# B&R Automation Studio project Sorting_Machine_DT
Automation Studio 4.9.2.46; technology packages: Acp10Arnc0 5.12.2, mappView 5.12.1

## Configuration Config1

CPU X20CP1584, AutomationRuntime C4.90, Build 4.1.2, Safety 0.0, Vc V4.72.2

### Task classes (Cpu.sw)
```
Cyclic#1 (cycle 2000 us, tolerance 0 us):
  X_AXIS_M <- XYZ_MANIPULATOR.X_AXIS_M.prg
  Y_AXIS_M <- XYZ_MANIPULATOR.Y_AXIS_M.prg
  Z_AXIS_M <- XYZ_MANIPULATOR.Z_AXIS_M.prg
  X_AXIS_CC <- CAMERA_CONVEYOR.X_AXIS_CC.prg
Cyclic#2 (cycle 10000 us, tolerance 10000 us):
  Main <- Main_Control.Main.prg
DataObjects: Acp10sys
NcDataObjects: acp10etxen <- Motion_Package.acp10etxen.dob, gAxis01_Xa <- Motion_Package.gAxis01_Xobj.gAxis01_Xa.dob, gAxis01_Xi <- Motion_Package.gAxis01_Xobj.gAxis01_Xi.dob, gAxis01_Ya <- Motion_Package.gAxis01_Yobj.gAxis01_Ya.dob, gAxis01_Yi <- Motion_Package.gAxis01_Yobj.gAxis01_Yi.dob, gAxis01_Za <- Motion_Package.gAxis01_Zobj.gAxis01_Za.dob, gAxis01_Zi <- Motion_Package.gAxis01_Zobj.gAxis01_Zi.dob, gAxis01_Ca <- Motion_Package.gAxis01_Cobj.gAxis01_Ca.dob, gAxis01_Ci <- Motion_Package.gAxis01_Cobj.gAxis01_Ci.dob
Binaries: udbdef, arsvcreg, FWRules, mvLoader, TCData, acp10cfg, Acp10map, iomap, asfw, Role, Config, sysconf, arconfig, ashwd, User, ashwac
Libraries: Acp10man, Acp10par, NcGlobal, Acp10_MC, sys_lib, brsystem, runtime, MpAxis, MpBase, MpCom, rp_funcx, standard, Acp10sim, astime, arssl, asbrstr, fileio, powerlnk, dataobj
```

### Hardware
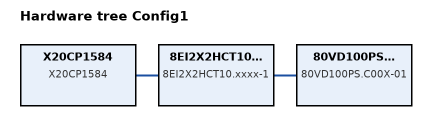
```
80VD100PS.C00X-01 : 80VD100PS.C00X-01 v2.5.0.0  [PLK1 -> 8EI2X2HCT10.xxxx-1.PLK2 (NodeNumber=2) [Cable Type=PowerlinkCable, Length=10, Version=1.0.0.3]]
  MotionTP = Acp10Arnc0
  Simulate = complete
  BothEndSwitchesAreNormallyOpen_r1 = on
  QuickStopIsNormallyOpen_r1 = on
8EI2X2HCT10.xxxx-1 : 8EI2X2HCT10.xxxx-1 v2.3.0.3  [PLK1 -> X20CP1584.IF3 (NodeNumber=1) [Cable Type=PowerlinkCable, Length=10, Version=1.0.0.3]; PLK2 -> 80VD100PS.C00X-01.PLK1 (NodeNumber=1) [Cable Type=PowerlinkCable, Length=10, Version=1.0.0.3]]
  MotionTP = Acp10Arnc0
  Simulate = complete
  BothEndSwitchesAreNormallyOpen_r1 = on
  QuickStopIsNormallyOpen_r1 = on
X20CP1584 : X20CP1584 v1.9.0.0
  Connector IF2:
    ActivateDevice = 1
  ConfigurationID = Sorting_Machine_DT_Config1
  Simulation = 1
  TimerDeviceType = EPLX2X
  TimerDevice = X20CP1584.IF3
  TaskClassIdleTime = 2000
  Cyclic1Duration = 2000
  Cyclic1Tolerance = 0
  Cyclic2Duration = 10000
  Cyclic2Tolerance = 10000
  ActivateOpcUa = 1
  OpcUaInformationModels_PV_Version = 1
```

### OpcUa.uanodeset - X20CP1584/Connectivity/OpcUA/OpcUa.uanodeset
```
UANodeSet:
  NamespaceUris:
    Uri = http://customer.com/mynamespace/
  Aliases:
    Alias = i=1 (Alias=Boolean)
    Alias = i=2 (Alias=SByte)
    Alias = i=3 (Alias=Byte)
    Alias = i=4 (Alias=Int16)
    Alias = i=5 (Alias=UInt16)
    Alias = i=6 (Alias=Int32)
    Alias = i=7 (Alias=UInt32)
    Alias = i=12 (Alias=String)
```

### Acp10cfg.ncc - X20CP1584/Motion/Acp10cfg.ncc
```
NcConfiguration (Version=5.12.2, NcSwId=Acp10)
  ACP10CF1_typ:
    cnt_nettrc_rec_drive = 1500
    bufsize_trace_upload = 1200
    tc_nc_man_task = Cyclic #1
    glob_pv_as_ncobject = Yes
    ncsys_dl_broadcast = Yes
    ncsys_dl_acp_reset = Yes
    safemc_log_err_to_ax = Yes
    network_init:
      ncsw_init_execute = Yes
      automatic_execute = No
      node_nr_warning = Yes
      net_err_before_ncact = Yes
    nettrc:
      enter_parsecrec = Yes
      enter_ncaction = Yes
      save_ring_startidx = Yes
    cam_prof_download:
      cam_dat_dl_parallel = No
      tc_cam_dl_parallel = Task class for NC Manager task
    plk_if[0]:
      if_name = IF3
      tc_CycDat_PLCopen = Task class for NC Manager task
      mc_broadcast_extdat = No
```

### Acp10map.ncm - X20CP1584/Motion/Acp10map.ncm
```
NcMapping (NcSwId=Acp10)
  NcObject gAxis01_X (ModuleId=8EI2X2HCT10.xxxx-1, Type=ncAXIS, Channel=1, AcoposSimulation=Off, InitParameter=gAxis01_Xi, AcoposParameter=gAxis01_Xa, Disabled=FALSE, ModuleDisabled=FALSE)
  NcObject gAxis01_Y (ModuleId=8EI2X2HCT10.xxxx-1, Type=ncAXIS, Channel=2, AcoposSimulation=Off, InitParameter=gAxis01_Yi, AcoposParameter=gAxis01_Ya, Disabled=FALSE, ModuleDisabled=FALSE)
  NcObject gAxis01_Z (ModuleId=8EI2X2HCT10.xxxx-1, Type=ncAXIS, Channel=3, AcoposSimulation=Off, InitParameter=gAxis01_Zi, AcoposParameter=gAxis01_Za, Disabled=FALSE, ModuleDisabled=FALSE)
  NcObject 8EI2X2HCT10.xxxx-1_ncV_AXIS1 (ModuleId=8EI2X2HCT10.xxxx-1, Type=ncV_AXIS, Channel=1, Disabled=TRUE, ModuleDisabled=FALSE)
  NcObject 8EI2X2HCT10.xxxx-1_ncV_AXIS2 (ModuleId=8EI2X2HCT10.xxxx-1, Type=ncV_AXIS, Channel=2, Disabled=TRUE, ModuleDisabled=FALSE)
  NcObject 8EI2X2HCT10.xxxx-1_ncV_AXIS3 (ModuleId=8EI2X2HCT10.xxxx-1, Type=ncV_AXIS, Channel=3, Disabled=TRUE, ModuleDisabled=FALSE)
  NcObject gAxis01_C (ModuleId=80VD100PS.C00X-01, Type=ncAXIS, Channel=1, AcoposSimulation=Off, InitParameter=gAxis01_Ci, AcoposParameter=gAxis01_Ca, Disabled=FALSE, ModuleDisabled=FALSE)
  NcObject 80VD100PS.C00X-01_ncV_AXIS1 (ModuleId=80VD100PS.C00X-01, Type=ncV_AXIS, Channel=1, Disabled=TRUE, ModuleDisabled=FALSE)
```

### Config.mpaxisbasic - X20CP1584/Motion/Config.mpaxisbasic
```
Element gAxisBasic_Axis_M_X (Type=mpaxisbasic)
Element gAxisBasic_Axis_M_Z (Type=mpaxisbasic)
Element gAxisBasic_Axis_M_Y (Type=mpaxisbasic)
Element gAxisBasic_Axis_CC_X (Type=mpaxisbasic)
```

- Safety project (password-protected, skipped)

## Logical view

Binary libraries used (declarations not repeated): operator, runtime, astime, AsIecCon, Acp10man 5.12.2, Acp10par 5.12.2, NcGlobal 5.12.2, Acp10_MC 5.12.2, sys_lib, brsystem, MpAxis 1.75.0, MpBase 5.12.0, MpCom 5.12.0, standard, Acp10sim 5.12.2

### Global.typ - Global data types
```iecst
TYPE
	mapp_view_str : 	STRUCT
		active : BOOL;
		is_homed : BOOL;
		power_on : BOOL;
		cam_obj_id : USINT;
		br_pad_obj_id : ARRAY[0..3]OF USINT;
		smc_pad_obj_id : ARRAY[0..3]OF USINT;
	END_STRUCT;
	object_str : 	STRUCT
		write : object_w_str;
		read : object_r_str;
	END_STRUCT;
	object_w_str : 	STRUCT
		set_object_id : USINT;
		reset : BOOL;
		detach : BOOL;
		attach : BOOL;
	END_STRUCT;
	object_r_str : 	STRUCT
		object_id : USINT;
		object_type : USINT;
	END_STRUCT;
	digT_service_control_str : 	STRUCT
		power : BOOL;
		home : BOOL;
		start : BOOL;
		actual_state : USINT;
		object : object_str;
		mapp_view : mapp_view_str;
	END_STRUCT;
	digT_control_llinp_str : 	STRUCT
		pos : LREAL;
		vel : LREAL;
	END_STRUCT;
	digT_control_linp_enum :
		(
		LINP_CTRL_WAIT_STATE := 0,
		LINP_CTRL_LOAD_PARAM_STATE := 10,
		LINP_CTRL_SET_POSITION_STATE := 11,
		LINP_CTRL_STOP_STATE := 12
		);
	axis_str : 	STRUCT
		actual_velocity : LREAL;
		actual_position : LREAL;
		actual_state : digT_control_linp_enum;
		parameter : digT_control_llinp_str;
		start : BOOL;
		stop : BOOL;
		active : BOOL;
		power_on : BOOL;
		is_homed : BOOL;
	END_STRUCT;
	camera_conv_str : 	STRUCT
		X : axis_str;
	END_STRUCT;
	xyz_manip_str : 	STRUCT
		X : axis_str;
		Y : axis_str;
		Z : axis_str;
	END_STRUCT;
	dt_main_str : 	STRUCT
		camera : camera_str;
		xyz_manipulator : xyz_manip_str;
		camera_conveyor : camera_conv_str;
		service : digT_service_control_str;
	END_STRUCT;
	camera_str : 	STRUCT
		scan : BOOL;
	END_STRUCT;
END_TYPE
```

### Global.var - Global variables
```iecst
VAR
	gAxis01_X : ACP10AXIS_typ;
	gAxis01_Y : ACP10AXIS_typ;
	gAxis01_Z : ACP10AXIS_typ;
	gAxis01_C : ACP10AXIS_typ;
	dT_Main : dt_main_str;
END_VAR
```

### Package Logical/Libraries - Global libraries

### Library Logical/Libraries/rp_funcx (ANSIC)

#### Types.typ - Exported data types
```iecst
TYPE
	default_param_smcT_str : 	STRUCT
		MAX_POSITION : LREAL;
		MIN_POSITION : LREAL;
		MAX_VELOCITY : LREAL;
		MIN_VELOCITY : LREAL;
	END_STRUCT;
	param_lim_struct : 	STRUCT
		velocity : LREAL;
		position_end : LREAL;
		position_start : LREAL;
		mode : limit_sequence_enum;
		time : ARRAY[0..1]OF TIME;
		signal : BOOL;
		signal_inPos : ARRAY[0..1]OF BOOL;
		elapsed_time : ARRAY[0..1]OF TIME;
		time_signal : ARRAY[0..1]OF USINT;
	END_STRUCT;
	parameters_structure_set : 	STRUCT
		position : LREAL;
		velocity : LREAL;
		limit : param_lim_struct;
		sequence : param_sv_struct;
		MAX_VELOCITY : LREAL := 0;
		MIN_VELOCITY : LREAL := 0;
		MAX_POSITION : LREAL := 0;
		MIN_POSITION : LREAL := 0;
		default_parameters : BOOL;
		set_velocity : LREAL;
		set_position : LREAL;
	END_STRUCT;
	parameters_structure_actual : 	STRUCT
		position : LREAL;
		velocity : REAL;
		torque : LREAL;
		motorTemperature : LREAL;
		lagError : LREAL;
		profinet_pos : ARRAY[0..5]OF USINT;
		profinet_vel : ARRAY[0..5]OF USINT;
	END_STRUCT;
	param_sv_struct : 	STRUCT
		position : ARRAY[0..4]OF LREAL;
		velocity : ARRAY[0..4]OF LREAL;
		mode : limit_sequence_enum;
		signal : BOOL;
		time : ARRAY[0..4]OF TIME;
		signal_inPos : ARRAY[0..4]OF BOOL;
		elapsed_time : ARRAY[0..4]OF TIME;
		time_signal : ARRAY[0..4]OF USINT;
	END_STRUCT;
	mode_structure : 	STRUCT
		manual : instruction_structure_manual;
		automatic : instruction_structure_auto;
		stop : BOOL;
		home : BOOL;
		mode : USINT;
	END_STRUCT;
	SMCTrak_enum :
		(
		INITIALIZATION_STATE := 0,
		POWER_STATE := 10,
		HOME_STATE_1 := 20,
		HOME_STATE_2 := 21,
		HOME_STATE_3 := 22,
		WAIT_STATE := 30,
		MOVE_HOME_1 := 35,
		MOVE_HOME_2 := 36,
		AUTO_MODE_STATE_RT_1 := 40,
		AUTO_MODE_STATE_RT_2 := 41,
		AUTO_MODE_STATE_RT_3 := 42,
		AUTO_MODE_STATE_UL_1 := 50,
		AUTO_MODE_STATE_UL_2 := 51,
		AUTO_MODE_STATE_UL_3 := 52,
		AUTO_MODE_STATE_SS_1 := 60,
		AUTO_MODE_STATE_SS_2 := 62,
		MANUAL_MODE_STATE_1 := 70,
		MANUAL_MODE_STATE_2 := 71,
		ERROR_STATE_1 := 100,
		ERROR_STATE_2 := 101,
		ERROR_STATE_3 := 102,
		ERROR_STATE_4 := 103,
		ERROR_STATE_5 := 104
		);
	limit_sequence_enum :
		(
		INSTR_SIGNAL := 0,
		INSTR_TIME := 1
		);
	Internal_structure_SMCtrak : 	STRUCT
		Before_state : SMCTrak_enum;
		State : SMCTrak_enum;
		Local : internal_local_smctrak;
		Timer : internal_smctrak_timer;
	END_STRUCT;
	internal_smctrak_timer : 	STRUCT
		enable_time : BOOL;
		output_time : BOOL;
		wait_time : TIME;
		elapsed_time : {REDUND_UNREPLICABLE} TIME;
	END_STRUCT;
	internal_local_smctrak : 	STRUCT
		set_position : LREAL;
		set_velocity : LREAL;
		before_position : LREAL;
		before_velocity : LREAL;
		sum_position : LREAL;
		sum_velocity : LREAL;
		count_sequence : USINT;
		pos_sequence : LREAL;
	END_STRUCT;
	instruction_structure_manual : 	STRUCT
		start : BOOL;
	END_STRUCT;
	instruction_structure_auto : 	STRUCT
		start : BOOL;
		instruction : automatic_instruction_enum;
	END_STRUCT;
	automatic_instruction_enum :
		(
		INSTR_REAL_TIME := 0,
		INSTR_LOWER_UPPER_LIMIT := 1,
		INSTR_SEQUENCE := 2
		);
END_TYPE
```

#### rp_funcx.fun - Exported functions and function blocks
```iecst
FUNCTION_BLOCK SMC_PAD (*TODO: Add your comment here*) (*$GROUP=User,$CAT=User,$GROUPICON=User.png,$CATICON=User.png*)
	VAR_INPUT
		Enable : {REDUND_UNREPLICABLE} BOOL;
		Power : BOOL;
		Home : BOOL;
		Absolute_Position : LREAL;
		MpAxis : REFERENCE TO MpAxisBasic;
		MpAxisParType : REFERENCE TO MpAxisBasicParType;
		MpAxisCyclic : REFERENCE TO MpAxisCyclicSet;
		MpAxisCyclicParType : REFERENCE TO MpAxisCyclicSetParType;
		Mode : mode_structure;
		Default_parameters : default_param_smcT_str;
		Set_Parameters : parameters_structure_set;
	END_VAR
	VAR_OUTPUT
		Actual_State : SMCTrak_enum;
		PowerOn : BOOL;
		IsHomed : BOOL;
		Actual_Parameters : parameters_structure_actual;
		InPosition : BOOL;
		Active : BOOL;
		Status : DINT;
	END_VAR
	VAR
		Internal : Internal_structure_SMCtrak;
	END_VAR
END_FUNCTION_BLOCK
```

#### SMC_PAD.c
```c
/**
 * MIT License
 * Copyright(c) 2020 Roman Parak
 * Permission is hereby granted, free of charge, to any person obtaining a copy
 * of this software and associated documentation files (the "Software"), to deal
 * in the Software without restriction, including without limitation the rights
 * to use, copy, modify, merge, publish, distribute, sublicense, and/or sell
 * copies of the Software, and to permit persons to whom the Software is
 * furnished to do so, subject to the following conditions:
 * The above copyright notice and this permission notice shall be included in all
 * copies or substantial portions of the Software.
 * THE SOFTWARE IS PROVIDED "AS IS", WITHOUT WARRANTY OF ANY KIND, EXPRESS OR
 * IMPLIED, INCLUDING BUT NOT LIMITED TO THE WARRANTIES OF MERCHANTABILITY,
 * FITNESS FOR A PARTICULAR PURPOSE AND NONINFRINGEMENT. IN NO EVENT SHALL THE
 * AUTHORS OR COPYRIGHT HOLDERS BE LIABLE FOR ANY CLAIM, DAMAGES OR OTHER
 * LIABILITY, WHETHER IN AN ACTION OF CONTRACT, TORT OR OTHERWISE, ARISING FROM,
 * OUT OF OR IN CONNECTION WITH THE SOFTWARE OR THE USE OR OTHER DEALINGS IN THE
 * SOFTWARE.
 */
/**
 * Author   : Roman Parak
 * Email    : Roman.Parak@outlook.com
 * File Name: SMC_PAD.c
 */

#include <bur/plctypes.h>
#include <stdio.h>
#include <stdlib.h>
#include <MpAxis.h>
#include <math.h>
#include <standard.h>

#ifdef __cplusplus
	extern "C"
	{
#endif
#include "rp_funcx.h"
#ifdef __cplusplus
	};
#endif

// ************************************************************************************************************************************ //
// -------------------------------------------------------------  DECLARATIONS -------------------------------------------------------- //
// ************************************************************************************************************************************ //
// Timer
_LOCAL TON_typ ton_1;
// FUNCTION // DECLARATION //
void update_cyclicParameters(struct SMC_PAD* smc_pad, LREAL position, LREAL velocity);
BOOL set_time(BOOL enable, TIME t);
// INITIALIZATION // RESET //
void initialization_smc_pad(struct SMC_PAD* smc_pad);
void reset_parameters(struct SMC_PAD* smc_pad);
void parameters_null(struct SMC_PAD* smc_pad);

// ************************************************************************************************************************************ //
// --------------------------------------------------------------  MAIN --------------------------------------------------------------- //
// ************************************************************************************************************************************ //
void SMC_PAD(struct SMC_PAD* smc_pad)
{
	// *********************************************************//
	// ---------------- INITIALIZATION  ----------------------- //
	// *********************************************************//
	if(smc_pad->Enable != 1){
		initialization_smc_pad(smc_pad);
	}

	// *********************************************************//
	// ---------------- PAD MAIN STATE  ----------------------- //
	// *********************************************************//
	switch(smc_pad->Internal.State){
		case INITIALIZATION_STATE:
			{
				/*************************************** INITIALIZATION STATE ******************************************/
				if((smc_pad->MpAxis->Error != 0 || smc_pad->MpAxisCyclic->Error != 0) || (smc_pad->MpAxis->StatusID != 0 || smc_pad->MpAxisCyclic->StatusID != 0)){
					smc_pad->Internal.Before_state = smc_pad->Internal.State;
					smc_pad->Internal.State 	   = ERROR_STATE_1;
				}

				if(smc_pad->MpAxis->Active == 1 && smc_pad->MpAxisCyclic->Active == 1){
					smc_pad->Active 	    = 1;
					smc_pad->Internal.State = POWER_STATE;
				}else{
					smc_pad->Active = 0;
				}
			}
			break;
		case POWER_STATE:
			{
				/*************************************** POWER STATE ******************************************/
				if((smc_pad->MpAxis->Error != 0 || smc_pad->MpAxisCyclic->Error != 0) || (smc_pad->MpAxis->StatusID != 0 || smc_pad->MpAxisCyclic->StatusID != 0)){
					smc_pad->Internal.Before_state = smc_pad->Internal.State;
					smc_pad->Internal.State 	   = ERROR_STATE_1;
				}

				if(smc_pad->Power == 1){
					// power state
					smc_pad->MpAxis->Power = 1;

					if(smc_pad->MpAxis->PowerOn == 1){
						smc_pad->Internal.State = HOME_STATE_1;
					}
				}
			}
			break;
		case HOME_STATE_1:
			{
				/*************************************** HOME (1) STATE ******************************************/
				if((smc_pad->MpAxis->Error != 0 || smc_pad->MpAxisCyclic->Error != 0) || (smc_pad->MpAxis->StatusID != 0 || smc_pad->MpAxisCyclic->StatusID != 0)){
					smc_pad->Internal.Before_state = smc_pad->Internal.State;
					smc_pad->Internal.State 	   = ERROR_STATE_1;
				}

				if(smc_pad->Home == 1){
					if(smc_pad->MpAxis->Position == 0 || (fabs(smc_pad->MpAxis->Position) == smc_pad->Absolute_Position)){
						// home state
						smc_pad->MpAxis->Home = 1;

						if(smc_pad->MpAxis->IsHomed == 1){
							smc_pad->MpAxis->Home   = 0;
							smc_pad->Internal.State = WAIT_STATE;
						}
					}else{
						smc_pad->Internal.State = HOME_STATE_2;
					}
				}

			}
			break;
		case HOME_STATE_2:
			{
				/*************************************** HOME (2) STATE ******************************************/
				if((smc_pad->MpAxis->Error != 0 || smc_pad->MpAxisCyclic->Error != 0) || (smc_pad->MpAxis->StatusID != 0 || smc_pad->MpAxisCyclic->StatusID != 0)){
					smc_pad->Internal.Before_state = smc_pad->Internal.State;
					smc_pad->Internal.State 	   = ERROR_STATE_1;
				}

				smc_pad->MpAxisParType->Home.Position = fabs(fabs(smc_pad->MpAxis->Position) - smc_pad->Absolute_Position);
				smc_pad->MpAxis->Update = 1;

				if(smc_pad->MpAxis->UpdateDone == 1){
					smc_pad->MpAxis->Update = 0;
					smc_pad->Internal.State = HOME_STATE_3;
				}

			}
			break;
		case HOME_STATE_3:
			{
				/*************************************** HOME (3) STATE ******************************************/
				if((smc_pad->MpAxis->Error != 0 || smc_pad->MpAxisCyclic->Error != 0) || (smc_pad->MpAxis->StatusID != 0 || smc_pad->MpAxisCyclic->StatusID != 0)){
					smc_pad->Internal.Before_state = smc_pad->Internal.State;
					smc_pad->Internal.State 	   = ERROR_STATE_1;
				}

				smc_pad->MpAxis->Home = 1;

				if(smc_pad->MpAxis->IsHomed == 1){
					smc_pad->MpAxis->Home   = 0;
					smc_pad->Internal.State = MOVE_HOME_1;
				}
			}
			break;
		case WAIT_STATE:
			{
				/*************************************** WAIT STATE ******************************************/
				if((smc_pad->MpAxis->Error != 0 || smc_pad->MpAxisCyclic->Error != 0) || (smc_pad->MpAxis->StatusID != 0 || smc_pad->MpAxisCyclic->StatusID != 0)){
					smc_pad->Internal.Before_state = smc_pad->Internal.State;
					smc_pad->Internal.State 	   = ERROR_STATE_1;
				}

				if(smc_pad->Mode.automatic.start == 1){
					smc_pad->MpAxis->Stop = 0;
					smc_pad->Mode.stop    = 0;
					if(smc_pad->Mode.automatic.instruction == INSTR_REAL_TIME){
						// real time {0}
						smc_pad->Internal.State  = AUTO_MODE_STATE_RT_1;
					}else if(smc_pad->Mode.automatic.instruction == INSTR_LOWER_UPPER_LIMIT){
						// upper / lower limit {1}
						// Set time parameters
						int i;
						for(i = 0; i < (int)(sizeof(smc_pad->Set_Parameters.limit.time)/sizeof(smc_pad->Set_Parameters.limit.time[0])); i++){
							if(smc_pad->Set_Parameters.limit.time_signal[i] == 0){
								smc_pad->Set_Parameters.limit.time[i] = 500;
							}else{
								smc_pad->Set_Parameters.limit.time[i] = smc_pad->Set_Parameters.limit.time_signal[0]*500;
							}
						}
						smc_pad->Internal.State  = AUTO_MODE_STATE_UL_1;
					}else if(smc_pad->Mode.automatic.instruction == INSTR_SEQUENCE){
						// sequence of steps {2}
						// Set time parameters
						int i;
						for(i = 0; i < (int)(sizeof(smc_pad->Set_Parameters.sequence.time)/sizeof(smc_pad->Set_Parameters.sequence.time[0])); i++){
							if(smc_pad->Set_Parameters.sequence.time_signal[i] == 0){
								smc_pad->Set_Parameters.sequence.time[i] = 500;
							}else{
								smc_pad->Set_Parameters.sequence.time[i] = smc_pad->Set_Parameters.sequence.time_signal[0]*500;
							}
						}
						smc_pad->Internal.State  = AUTO_MODE_STATE_SS_1;
					}
				}else if(smc_pad->Mode.manual.start == 1){
					smc_pad->Mode.stop      = 0;
					smc_pad->Internal.State = MANUAL_MODE_STATE_1;
				}else if(smc_pad->Mode.home == 1){
					if(smc_pad->MpAxisCyclic->Info.SlavePosition != 0){
						smc_pad->Internal.State = MOVE_HOME_1;
					}
				}else{
					smc_pad->Mode.stop = 0;
				}
			}
			break;
		case MOVE_HOME_1:
			{
				/*************************************** MOVE HOME (1) STATE ******************************************/
				if((smc_pad->MpAxis->Error != 0 || smc_pad->MpAxisCyclic->Error != 0) || (smc_pad->MpAxis->StatusID != 0 || smc_pad->MpAxisCyclic->StatusID != 0)){
					smc_pad->Internal.Before_state = smc_pad->Internal.State;
					smc_pad->Internal.State 	   = ERROR_STATE_1;
				}

				update_cyclicParameters(smc_pad, smc_pad->MpAxisCyclic->Info.SlavePosition, (smc_pad->Set_Parameters.MIN_VELOCITY*30));

				smc_pad->MpAxisCyclic->Update = 1;

				if(smc_pad->MpAxisCyclic->UpdateDone == 1){
					smc_pad->MpAxisCyclic->Update = 0;
					smc_pad->Internal.State       = MOVE_HOME_2;
				}
			}
			break;
		case MOVE_HOME_2:
			{
				/*************************************** MOVE HOME (2) STATE ******************************************/
				if((smc_pad->MpAxis->Error != 0 || smc_pad->MpAxisCyclic->Error != 0) || (smc_pad->MpAxis->StatusID != 0 || smc_pad->MpAxisCyclic->StatusID != 0)){
					smc_pad->Internal.Before_state = smc_pad->Internal.State;
					smc_pad->Internal.State 	   = ERROR_STATE_1;
				}

				if(smc_pad->MpAxisCyclic->CyclicPosition == 0){
					smc_pad->MpAxisCyclic->CyclicPosition = 1;
				}

				smc_pad->MpAxisCyclic->Position = smc_pad->Set_Parameters.MIN_POSITION;

				if(smc_pad->MpAxisCyclic->Info.SlavePosition == 0){
					smc_pad->Mode.home      = 0;
					smc_pad->Internal.State = WAIT_STATE;
				}
			}
			break;
		case AUTO_MODE_STATE_RT_1:
			{
				/*************************************** AUTO MODE Real-Time (1) STATE ******************************************/
				if((smc_pad->MpAxis->Error != 0 || smc_pad->MpAxisCyclic->Error != 0) || (smc_pad->MpAxis->StatusID != 0 || smc_pad->MpAxisCyclic->StatusID != 0)){
					smc_pad->Internal.Before_state = smc_pad->Internal.State;
					smc_pad->Internal.State 	   = ERROR_STATE_1;
				}

				if(smc_pad->Set_Parameters.position != smc_pad->Internal.Local.before_position){
					smc_pad->MpAxisCyclic->Position 	 = smc_pad->Set_Parameters.position;
					smc_pad->Internal.Local.set_position = smc_pad->Set_Parameters.position;
					smc_pad->Internal.Local.set_velocity = smc_pad->Set_Parameters.velocity;

					if((fabs(smc_pad->Set_Parameters.position - smc_pad->Internal.Local.before_position) == smc_pad->Internal.Local.sum_position) && (fabs(smc_pad->Set_Parameters.velocity - smc_pad->Internal.Local.before_velocity) == smc_pad->Internal.Local.sum_velocity)){
						smc_pad->Internal.State = AUTO_MODE_STATE_RT_2;
					}else{
						smc_pad->Internal.Local.sum_position  = fabs(smc_pad->Set_Parameters.position - smc_pad->Internal.Local.before_position);
						smc_pad->Internal.Local.sum_velocity  = fabs(smc_pad->Set_Parameters.velocity - smc_pad->Internal.Local.before_velocity);
						smc_pad->Internal.State         	  = AUTO_MODE_STATE_RT_3;
					}
				}
			}
			break;
		case AUTO_MODE_STATE_RT_2:
			{
				/*************************************** AUTO MODE Real-Time (2) STATE ******************************************/
				if((smc_pad->MpAxis->Error != 0 || smc_pad->MpAxisCyclic->Error != 0) || (smc_pad->MpAxis->StatusID != 0 || smc_pad->MpAxisCyclic->StatusID != 0)){
					smc_pad->Internal.Before_state = smc_pad->Internal.State;
					smc_pad->Internal.State 	   = ERROR_STATE_1;
				}

				if(smc_pad->MpAxisCyclic->CyclicPosition == 0){
					smc_pad->MpAxisCyclic->CyclicPosition = 1;
				}

				if(smc_pad->MpAxisCyclic->Info.SlavePosition == smc_pad->Internal.Local.set_position){
					smc_pad->Internal.Local.before_position = smc_pad->Internal.Local.set_position;
					smc_pad->Internal.Local.before_velocity = smc_pad->Internal.Local.set_velocity;
					smc_pad->Internal.State           	    = AUTO_MODE_STATE_RT_1;
				}
			}
			break;
		case AUTO_MODE_STATE_RT_3:
			{
				/*************************************** AUTO MODE Real-Time (3) STATE ******************************************/
				if((smc_pad->MpAxis->Error != 0 || smc_pad->MpAxisCyclic->Error != 0) || (smc_pad->MpAxis->StatusID != 0 || smc_pad->MpAxisCyclic->StatusID != 0)){
					smc_pad->Internal.Before_state = smc_pad->Internal.State;
					smc_pad->Internal.State 	   = ERROR_STATE_1;
				}

				update_cyclicParameters(smc_pad, fabs(smc_pad->Set_Parameters.position - smc_pad->MpAxisCyclic->Info.SlavePosition), smc_pad->Set_Parameters.velocity);

				smc_pad->MpAxisCyclic->Update = 1;

				if(smc_pad->MpAxisCyclic->UpdateDone == 1){
					smc_pad->MpAxisCyclic->Update = 0;
					smc_pad->Internal.State       = AUTO_MODE_STATE_RT_2;
				}
			}
			break;
		case MANUAL_MODE_STATE_1:
			{
				/*************************************** MANUAL MODE (1) STATE ******************************************/
				if((smc_pad->MpAxis->Error != 0 || smc_pad->MpAxisCyclic->Error != 0) || (smc_pad->MpAxis->StatusID != 0 || smc_pad->MpAxisCyclic->StatusID != 0)){
					smc_pad->Internal.Before_state = smc_pad->Internal.State;
					smc_pad->Internal.State 	   = ERROR_STATE_1;
				}

				update_cyclicParameters(smc_pad, smc_pad->Set_Parameters.MAX_POSITION, smc_pad->Set_Parameters.MAX_VELOCITY);

				smc_pad->MpAxisCyclic->Update = 1;

				if(smc_pad->MpAxisCyclic->UpdateDone == 1){
					smc_pad->MpAxisCyclic->Update = 0;
					smc_pad->Internal.State       = MANUAL_MODE_STATE_2;
				}
			}
			break;
		case MANUAL_MODE_STATE_2:
			{
				/*************************************** MANUAL MODE (2) STATE ******************************************/
				if((smc_pad->MpAxis->Error != 0 || smc_pad->MpAxisCyclic->Error != 0) || (smc_pad->MpAxis->StatusID != 0 || smc_pad->MpAxisCyclic->StatusID != 0)){
					smc_pad->Internal.Before_state = smc_pad->Internal.State;
					smc_pad->Internal.State 	   = ERROR_STATE_1;
				}

				if(smc_pad->MpAxisCyclic->CyclicPosition == 0){
					smc_pad->MpAxisCyclic->CyclicPosition = 1;
				}

				smc_pad->MpAxisCyclic->Position = smc_pad->Set_Parameters.position;
			}
			break;
		case AUTO_MODE_STATE_UL_1:
			{
				/*************************************** AUTO MODE Upper/Lower (1) STATE ******************************************/
				if((smc_pad->MpAxis->Error != 0 || smc_pad->MpAxisCyclic->Error != 0) || (smc_pad->MpAxis->StatusID != 0 || smc_pad->MpAxisCyclic->StatusID != 0)){
					smc_pad->Internal.Before_state = smc_pad->Internal.State;
					smc_pad->Internal.State 	   = ERROR_STATE_1;
				}

				update_cyclicParameters(smc_pad, (smc_pad->Set_Parameters.limit.position_start - smc_pad->Set_Parameters.limit.position_end), smc_pad->Set_Parameters.limit.velocity);

				smc_pad->MpAxisCyclic->Update = 1;

				if(smc_pad->MpAxisCyclic->UpdateDone == 1){
					smc_pad->MpAxisCyclic->Update = 0;
					smc_pad->Internal.State       = AUTO_MODE_STATE_UL_2;
				}
			}
			break;
		case AUTO_MODE_STATE_UL_2:
			{
				/*************************************** AUTO MODE Upper/Lower (2) STATE ******************************************/
				if((smc_pad->MpAxis->Error != 0 || smc_pad->MpAxisCyclic->Error != 0) || (smc_pad->MpAxis->StatusID != 0 || smc_pad->MpAxisCyclic->StatusID != 0)){
					smc_pad->Internal.Before_state = smc_pad->Internal.State;
					smc_pad->Internal.State 	   = ERROR_STATE_1;
				}

				if(smc_pad->MpAxisCyclic->CyclicPosition == 0){
					smc_pad->MpAxisCyclic->CyclicPosition = 1;
				}

				if(smc_pad->MpAxisCyclic->Info.SlavePosition != smc_pad->Set_Parameters.limit.position_start){
					smc_pad->MpAxisCyclic->Position = smc_pad->Set_Parameters.limit.position_start;
				}

				if(smc_pad->MpAxisCyclic->Info.SlavePosition == smc_pad->Set_Parameters.limit.position_start){
					if(smc_pad->Set_Parameters.limit.mode == INSTR_SIGNAL){
						smc_pad->Set_Parameters.limit.signal_inPos[0] = 1;
					}
					if(smc_pad->Set_Parameters.limit.mode == INSTR_SIGNAL && smc_pad->Set_Parameters.limit.signal == 1){
						// {SIGNAL}
						smc_pad->Internal.State  					  = AUTO_MODE_STATE_UL_3;
						smc_pad->Set_Parameters.limit.signal_inPos[0] = 0;
					}else if(smc_pad->Set_Parameters.limit.mode == INSTR_TIME){
						// {TIME}
						smc_pad->Internal.Timer.enable_time 		  = 1;
						smc_pad->Internal.Timer.wait_time   		  = smc_pad->Set_Parameters.limit.time[0];
						smc_pad->Set_Parameters.limit.elapsed_time[0] = smc_pad->Internal.Timer.elapsed_time;
						if(smc_pad->Internal.Timer.output_time == 1){
							smc_pad->Set_Parameters.limit.elapsed_time[0] = 0;
							smc_pad->Internal.Timer.enable_time   		  = 0;
							smc_pad->Internal.State 			  		  = AUTO_MODE_STATE_UL_3;
						}
					}
				}
			}
			break;
		case AUTO_MODE_STATE_UL_3:
			{
				/*************************************** AUTO MODE Upper/Lower (1) STATE ******************************************/
				if((smc_pad->MpAxis->Error != 0 || smc_pad->MpAxisCyclic->Error != 0) || (smc_pad->MpAxis->StatusID != 0 || smc_pad->MpAxisCyclic->StatusID != 0)){
					smc_pad->Internal.Before_state = smc_pad->Internal.State;
					smc_pad->Internal.State 	   = ERROR_STATE_1;
				}

				if(smc_pad->MpAxisCyclic->CyclicPosition == 0){
					smc_pad->MpAxisCyclic->CyclicPosition = 1;
				}

				smc_pad->MpAxisCyclic->Position = smc_pad->Set_Parameters.limit.position_end;

				if(smc_pad->MpAxisCyclic->Info.SlavePosition == smc_pad->Set_Parameters.limit.position_end){
					if(smc_pad->Set_Parameters.limit.mode == INSTR_SIGNAL){
						smc_pad->Set_Parameters.limit.signal_inPos[1] = 1;
					}
					if(smc_pad->Set_Parameters.limit.mode == INSTR_SIGNAL && smc_pad->Set_Parameters.limit.signal == 1){
						smc_pad->Set_Parameters.limit.signal_inPos[1] = 0;
						smc_pad->Internal.State 				      = AUTO_MODE_STATE_UL_2;
					}else if(smc_pad->Set_Parameters.limit.mode == INSTR_TIME){
						// {TIME}
						smc_pad->Internal.Timer.enable_time 		  = 1;
						smc_pad->Internal.Timer.wait_time   		  = smc_pad->Set_Parameters.limit.time[1];
						smc_pad->Set_Parameters.limit.elapsed_time[1] = smc_pad->Internal.Timer.elapsed_time;
						if(smc_pad->Internal.Timer.output_time == 1){
							smc_pad->Set_Parameters.limit.elapsed_time[1] = 0;
							smc_pad->Internal.Timer.enable_time   		  = 0;
							smc_pad->Internal.State 			  		  = AUTO_MODE_STATE_UL_2;
						}
					}
				}
			}
			break;
		case AUTO_MODE_STATE_SS_1:
			{
				/*************************************** AUTO MODE Sequence Step (1) STATE ******************************************/
				if((smc_pad->MpAxis->Error != 0 || smc_pad->MpAxisCyclic->Error != 0) || (smc_pad->MpAxis->StatusID != 0 || smc_pad->MpAxisCyclic->StatusID != 0)){
					smc_pad->Internal.Before_state = smc_pad->Internal.State;
					smc_pad->Internal.State 	   = ERROR_STATE_1;
				}

				update_cyclicParameters(smc_pad, (smc_pad->Set_Parameters.sequence.position[smc_pad->Internal.Local.count_sequence] - smc_pad->MpAxisCyclic->Info.SlavePosition), smc_pad->Set_Parameters.sequence.velocity[smc_pad->Internal.Local.count_sequence]);

				smc_pad->MpAxisCyclic->Update = 1;

				if(smc_pad->MpAxisCyclic->UpdateDone == 1){
					smc_pad->MpAxisCyclic->Update = 0;
					smc_pad->Internal.State       = AUTO_MODE_STATE_SS_2;
				}
			}
			break;
		case AUTO_MODE_STATE_SS_2:
			{
				/*************************************** AUTO MODE Sequence Step (2) STATE ******************************************/
				if((smc_pad->MpAxis->Error != 0 || smc_pad->MpAxisCyclic->Error != 0) || (smc_pad->MpAxis->StatusID != 0 || smc_pad->MpAxisCyclic->StatusID != 0)){
					smc_pad->Internal.Before_state = smc_pad->Internal.State;
					smc_pad->Internal.State 	   = ERROR_STATE_1;
				}

				if(smc_pad->MpAxisCyclic->CyclicPosition == 0){
					smc_pad->MpAxisCyclic->CyclicPosition = 1;
				}

				smc_pad->MpAxisCyclic->Position = smc_pad->Set_Parameters.sequence.position[smc_pad->Internal.Local.count_sequence];

				if(smc_pad->MpAxisCyclic->Info.SlavePosition == smc_pad->Set_Parameters.sequence.position[smc_pad->Internal.Local.count_sequence]){
					if(smc_pad->Set_Parameters.sequence.mode == INSTR_SIGNAL){
						smc_pad->Set_Parameters.sequence.signal_inPos[smc_pad->Internal.Local.count_sequence] = 1;
					}
					if(smc_pad->Set_Parameters.sequence.mode == INSTR_SIGNAL && smc_pad->Set_Parameters.sequence.signal == 1){
						// {SIGNAL}
						smc_pad->Set_Parameters.sequence.signal_inPos[smc_pad->Internal.Local.count_sequence] = 0;
						if(smc_pad->Internal.Local.count_sequence == 4){
							smc_pad->Internal.Local.count_sequence = 0;

							if(fabs(smc_pad->Set_Parameters.sequence.position[smc_pad->Internal.Local.count_sequence + 1] - smc_pad->MpAxisCyclic->Info.SlavePosition) != smc_pad->Internal.Local.pos_sequence){
								smc_pad->Internal.State = AUTO_MODE_STATE_SS_1;
							}
						}else{
							if(fabs(smc_pad->Set_Parameters.sequence.position[smc_pad->Internal.Local.count_sequence + 1] - smc_pad->MpAxisCyclic->Info.SlavePosition) != smc_pad->Internal.Local.pos_sequence){
								smc_pad->Internal.State = AUTO_MODE_STATE_SS_1;
							}
							smc_pad->Internal.Local.count_sequence++;
						}
					}else if(smc_pad->Set_Parameters.sequence.mode == INSTR_TIME){
						// {TIME}
						smc_pad->Internal.Timer.enable_time 												  = 1;
						smc_pad->Internal.Timer.wait_time  													  = smc_pad->Set_Parameters.sequence.time[smc_pad->Internal.Local.count_sequence];
						smc_pad->Set_Parameters.sequence.elapsed_time[smc_pad->Internal.Local.count_sequence] = smc_pad->Internal.Timer.elapsed_time;
						if(smc_pad->Internal.Timer.output_time == 1){
							smc_pad->Set_Parameters.sequence.elapsed_time[smc_pad->Internal.Local.count_sequence] = 0;
							smc_pad->Internal.Timer.enable_time 												  = 0;
							if(smc_pad->Internal.Local.count_sequence == 4){
								smc_pad->Internal.Local.count_sequence = 0;

								if(fabs(smc_pad->Set_Parameters.sequence.position[smc_pad->Internal.Local.count_sequence + 1] - smc_pad->MpAxisCyclic->Info.SlavePosition) != smc_pad->Internal.Local.pos_sequence){
									smc_pad->Internal.State = AUTO_MODE_STATE_SS_1;
								}
							}else{
								if(fabs(smc_pad->Set_Parameters.sequence.position[smc_pad->Internal.Local.count_sequence + 1] - smc_pad->MpAxisCyclic->Info.SlavePosition) != smc_pad->Internal.Local.pos_sequence){
									smc_pad->Internal.State = AUTO_MODE_STATE_SS_1;
								}
								smc_pad->Internal.Local.count_sequence++;
							}
						}
					}
				}

			}
			break;

		case ERROR_STATE_1:
			{
				/*************************************** ERROR (1) STATE ******************************************/
				if(smc_pad->MpAxisCyclic->CyclicPosition != 0){
					smc_pad->MpAxisCyclic->CyclicPosition = 0;
				}

				smc_pad->MpAxis->Stop = 0;

				if(smc_pad->MpAxis->Stopped == 0){
					smc_pad->Internal.State = ERROR_STATE_2;
				}

			}
			break;
		case ERROR_STATE_2:
			{
				/*************************************** ERROR (2) STATE ******************************************/
				smc_pad->MpAxis->Power = 0;

				if(smc_pad->MpAxis->PowerOn == 0){
					smc_pad->Internal.State = ERROR_STATE_3;
				}

			}
			break;
		case ERROR_STATE_3:
			{
				/*************************************** ERROR (3) STATE ******************************************/
				smc_pad->MpAxisCyclic->ErrorReset = 1;

				if(smc_pad->MpAxisCyclic->Error == 0 && smc_pad->MpAxisCyclic->StatusID == 0){
					smc_pad->MpAxisCyclic->ErrorReset = 0;
					smc_pad->Internal.State           = ERROR_STATE_4;
				}
			}
			break;
		case ERROR_STATE_4:
			{
				/*************************************** ERROR (4) STATE ******************************************/
				smc_pad->MpAxis->ErrorReset 	  = 1;

				if(smc_pad->MpAxis->Error == 0 && smc_pad->MpAxis->StatusID == 0){
					smc_pad->MpAxis->ErrorReset = 0;
					if(smc_pad->Power == 1){
						smc_pad->Internal.State = ERROR_STATE_5;
					}else{
						smc_pad->Internal.State = smc_pad->Internal.Before_state;
					}
				}
			}
			break;
		case ERROR_STATE_5:
			{
				/*************************************** ERROR (5) STATE ******************************************/
				smc_pad->MpAxis->Power = 1;

				if((smc_pad->MpAxis->Error != 0 || smc_pad->MpAxisCyclic->Error != 0) || (smc_pad->MpAxis->StatusID != 0 || smc_pad->MpAxisCyclic->StatusID != 0)){
					smc_pad->Internal.State 	   = ERROR_STATE_1;
				}

				if(smc_pad->MpAxis->PowerOn == 1){
					smc_pad->MpAxisCyclic->CyclicPosition = 1;
					smc_pad->Internal.State               = smc_pad->Internal.Before_state;
				}
			}
			break;

	} // end switch

	// **************** STOP MODE SMC PAD **********************//
	if(smc_pad->Mode.stop == 1){
		// Mapp axis
		smc_pad->MpAxisCyclic->CyclicPosition = 0;
		smc_pad->MpAxis->Stop                 = 1;

		parameters_null(smc_pad);

		if(smc_pad->MpAxis->Stopped == 1){
			// state
			smc_pad->Internal.State = WAIT_STATE;
		}
	}

	//********************** BORDER CONTROLS **********************//
	if(smc_pad->Mode.automatic.start == 1 || smc_pad->Mode.manual.start == 1){
		if(smc_pad->Mode.automatic.instruction == INSTR_REAL_TIME){
			// Automatic/Manual {position}
			if(smc_pad->Set_Parameters.position > smc_pad->Set_Parameters.MAX_POSITION){
				smc_pad->Set_Parameters.position = smc_pad->Set_Parameters.MAX_POSITION;
			}else if(smc_pad->Set_Parameters.position < smc_pad->Set_Parameters.MIN_POSITION){
				smc_pad->Set_Parameters.position = smc_pad->Set_Parameters.MIN_POSITION;
			}

			// Automatic/Manual {velocity}
			if(smc_pad->Set_Parameters.velocity > smc_pad->Set_Parameters.MAX_VELOCITY){
				smc_pad->Set_Parameters.velocity  = smc_pad->Set_Parameters.MAX_VELOCITY;
			}else if(smc_pad->Set_Parameters.velocity < smc_pad->Set_Parameters.MIN_VELOCITY){
				smc_pad->Set_Parameters.velocity  = smc_pad->Set_Parameters.MIN_VELOCITY;
			}
		}
	}

	if(smc_pad->Mode.automatic.start == 1 && smc_pad->Mode.automatic.instruction == INSTR_LOWER_UPPER_LIMIT){
		// Limit {position}
		if(smc_pad->Set_Parameters.limit.position_end > smc_pad->Set_Parameters.MAX_POSITION){
			smc_pad->Set_Parameters.limit.position_end = smc_pad->Set_Parameters.MAX_POSITION;
		}else if(smc_pad->Set_Parameters.limit.position_start < smc_pad->Set_Parameters.MIN_POSITION){
			smc_pad->Set_Parameters.limit.position_start = smc_pad->Set_Parameters.MIN_POSITION;
		}
		// Limit {velocity}
		if(smc_pad->Set_Parameters.limit.velocity > smc_pad->Set_Parameters.MAX_VELOCITY){
			smc_pad->Set_Parameters.limit.velocity = smc_pad->Set_Parameters.MAX_VELOCITY;
		}else if(smc_pad->Set_Parameters.limit.velocity < smc_pad->Set_Parameters.MIN_VELOCITY){
			smc_pad->Set_Parameters.limit.velocity  = smc_pad->Set_Parameters.MIN_VELOCITY;
		}
	}

	if(smc_pad->Mode.automatic.start == 1 && smc_pad->Mode.automatic.instruction == INSTR_SEQUENCE){
		// Sequence {position}
		int i_pos;
		for(i_pos = 0; i_pos < 5; i_pos++){
			if(smc_pad->Set_Parameters.sequence.position[i_pos] > smc_pad->Set_Parameters.MAX_POSITION){
				smc_pad->Set_Parameters.sequence.position[i_pos] = smc_pad->Set_Parameters.MAX_POSITION;
			}else if(smc_pad->Set_Parameters.sequence.position[i_pos] < smc_pad->Set_Parameters.MIN_POSITION){
				smc_pad->Set_Parameters.sequence.position[i_pos] = smc_pad->Set_Parameters.MIN_POSITION;
			}
		}
		// Sequence {velocity}
		int i_vel;
		for(i_vel = 0; i_vel < 5; i_vel++){
			if(smc_pad->Set_Parameters.sequence.velocity[i_vel] > smc_pad->Set_Parameters.MAX_POSITION){
				smc_pad->Set_Parameters.sequence.velocity[i_vel] = smc_pad->Set_Parameters.MAX_POSITION;
			}else if(smc_pad->Set_Parameters.sequence.velocity[i_vel] < smc_pad->Set_Parameters.MIN_POSITION){
				smc_pad->Set_Parameters.sequence.velocity[i_vel] = smc_pad->Set_Parameters.MIN_POSITION;
			}
		}
	}

	//**************** OUTPUT VARIABLES **********************//
	// SMC PAD
	smc_pad->Actual_Parameters.position 		= smc_pad->MpAxisCyclic->Info.SlavePosition;
	smc_pad->Actual_Parameters.velocity 		= smc_pad->MpAxisCyclic->Info.SlaveVelocity;
	smc_pad->Actual_Parameters.lagError 		= smc_pad->MpAxis->Info.CyclicRead.LagError.Value;
	smc_pad->Actual_Parameters.motorTemperature = smc_pad->MpAxis->Info.CyclicRead.MotorTemperature.Value;
	smc_pad->Actual_Parameters.torque  			= smc_pad->MpAxis->Info.CyclicRead.Torque.Value;

	smc_pad->Set_Parameters.set_position = smc_pad->MpAxisCyclic->Position;
	if(smc_pad->MpAxis->Velocity >= 0){
		smc_pad->Set_Parameters.set_velocity = smc_pad->MpAxisCyclicParType->PositionModeMaxVelocity;
	}else{
		smc_pad->Set_Parameters.set_velocity = (-1)*smc_pad->MpAxisCyclicParType->PositionModeMaxVelocity;
	}

	smc_pad->PowerOn      = smc_pad->MpAxis->PowerOn;
	smc_pad->IsHomed      = smc_pad->MpAxis->IsHomed;
	smc_pad->Actual_State = smc_pad->Internal.State;
	smc_pad->Status       = smc_pad->MpAxis->StatusID;
	smc_pad->InPosition   = smc_pad->MpAxis->InPosition;

	// Set default parameters
	if(smc_pad->Set_Parameters.default_parameters == 1){
		smc_pad->Set_Parameters.MAX_POSITION = smc_pad->Default_parameters.MAX_POSITION;
		smc_pad->Set_Parameters.MIN_POSITION = smc_pad->Default_parameters.MIN_POSITION;
		smc_pad->Set_Parameters.MAX_VELOCITY = smc_pad->Default_parameters.MAX_VELOCITY;
		smc_pad->Set_Parameters.MIN_VELOCITY = smc_pad->Default_parameters.MIN_VELOCITY;
	}
	// Parameters - round function
	smc_pad->Set_Parameters.position = round(smc_pad->Set_Parameters.position);
	smc_pad->Set_Parameters.velocity = round(smc_pad->Set_Parameters.velocity);
	smc_pad->Set_Parameters.limit.position_start = round(smc_pad->Set_Parameters.limit.position_start);
	smc_pad->Set_Parameters.limit.position_end   = round(smc_pad->Set_Parameters.limit.position_end);
	smc_pad->Set_Parameters.limit.velocity       = round(smc_pad->Set_Parameters.limit.velocity);
	smc_pad->Set_Parameters.sequence.position[0] = round(smc_pad->Set_Parameters.sequence.position[0]);
	smc_pad->Set_Parameters.sequence.position[1] = round(smc_pad->Set_Parameters.sequence.position[1]);
	smc_pad->Set_Parameters.sequence.position[2] = round(smc_pad->Set_Parameters.sequence.position[2]);
	smc_pad->Set_Parameters.sequence.position[3] = round(smc_pad->Set_Parameters.sequence.position[3]);
	smc_pad->Set_Parameters.sequence.position[4] = round(smc_pad->Set_Parameters.sequence.position[4]);
	smc_pad->Set_Parameters.sequence.velocity[0] = round(smc_pad->Set_Parameters.sequence.velocity[0]);
	smc_pad->Set_Parameters.sequence.velocity[1] = round(smc_pad->Set_Parameters.sequence.velocity[1]);
	smc_pad->Set_Parameters.sequence.velocity[2] = round(smc_pad->Set_Parameters.sequence.velocity[2]);
	smc_pad->Set_Parameters.sequence.velocity[3] = round(smc_pad->Set_Parameters.sequence.velocity[3]);
	smc_pad->Set_Parameters.sequence.velocity[4] = round(smc_pad->Set_Parameters.sequence.velocity[4]);

	// *********************************************************//
	// -------------------- CALL FUNCTIONS -------------------- //
	// *********************************************************//
	// Set wait time {Global}
	if(smc_pad->Set_Parameters.limit.mode == INSTR_TIME || smc_pad->Set_Parameters.sequence.mode == INSTR_TIME){
		smc_pad->Internal.Timer.output_time  = set_time(smc_pad->Internal.Timer.enable_time, smc_pad->Internal.Timer.wait_time);
		smc_pad->Internal.Timer.elapsed_time = ton_1.ET;
	}
}// end function block

// ************************************************************************************************************************************ //
// ------------------------------------------------------------  FUNCTIONS ------------------------------------------------------------ //
// ************************************************************************************************************************************ //

// ****************INITIALIZATION PARAMETERS **********************//
void initialization_smc_pad(struct SMC_PAD* smc_pad)
{
	// initialization state
	smc_pad->Internal.State 	   = INITIALIZATION_STATE;
	smc_pad->Internal.Before_state = INITIALIZATION_STATE;
	// reset parameters
	reset_parameters(smc_pad);

} // end function

// ****************RESET PARAMETERS **********************//
void reset_parameters(struct SMC_PAD* smc_pad){
	// Power & Home {Input}
	smc_pad->Power = 0;
	smc_pad->Home  = 0;
	// Parameters {Input}
	smc_pad->Absolute_Position 			 = 0;
	// Parameters Mode structure {Input}
	smc_pad->Mode.home = 0;
	smc_pad->Mode.stop = 0;
	// Mode {automatic}
	smc_pad->Mode.automatic.instruction = INSTR_REAL_TIME;
	smc_pad->Mode.automatic.start       = 0;
	// Mode {manual}
	smc_pad->Mode.manual.start          = 0;
	// Set parameters structure {Input}
	smc_pad->Set_Parameters.position = 0;
	smc_pad->Set_Parameters.velocity = 0;
	// Set parameters {limit}
	smc_pad->Set_Parameters.limit.mode = INSTR_SIGNAL;
	smc_pad->Set_Parameters.limit.position_end   = 0;
	smc_pad->Set_Parameters.limit.position_start = 0;
	smc_pad->Set_Parameters.limit.signal         = 0;
	smc_pad->Set_Parameters.limit.time[0]        = 0;
	smc_pad->Set_Parameters.limit.time[1]        = 0;
	smc_pad->Set_Parameters.limit.velocity       = 0;
	// Signal {limit/in position}
	smc_pad->Set_Parameters.limit.signal_inPos[0] = 0;
	smc_pad->Set_Parameters.limit.signal_inPos[1] = 0;
	// Set parameters {sequence}
	smc_pad->Set_Parameters.sequence.mode = INSTR_SIGNAL;
	// Set parameters {sequence/position}
	smc_pad->Set_Parameters.sequence.position[0] = 0;
	smc_pad->Set_Parameters.sequence.position[1] = 0;
	smc_pad->Set_Parameters.sequence.position[2] = 0;
	smc_pad->Set_Parameters.sequence.position[3] = 0;
	smc_pad->Set_Parameters.sequence.position[4] = 0;
	// Set parameters {sequence/velocity}
	smc_pad->Set_Parameters.sequence.velocity[0] = 0;
	smc_pad->Set_Parameters.sequence.velocity[1] = 0;
	smc_pad->Set_Parameters.sequence.velocity[2] = 0;
	smc_pad->Set_Parameters.sequence.velocity[3] = 0;
	smc_pad->Set_Parameters.sequence.velocity[4] = 0;
	// Set parameters {sequence/time}
	smc_pad->Set_Parameters.sequence.time[0] = 0;
	smc_pad->Set_Parameters.sequence.time[1] = 0;
	smc_pad->Set_Parameters.sequence.time[2] = 0;
	smc_pad->Set_Parameters.sequence.time[3] = 0;
	smc_pad->Set_Parameters.sequence.time[4] = 0;
	// Signal {sequence/in position}
	smc_pad->Set_Parameters.sequence.signal_inPos[0] = 0;
	smc_pad->Set_Parameters.sequence.signal_inPos[1] = 0;
	smc_pad->Set_Parameters.sequence.signal_inPos[2] = 0;
	smc_pad->Set_Parameters.sequence.signal_inPos[3] = 0;
	smc_pad->Set_Parameters.sequence.signal_inPos[4] = 0;
	// Actual parameters structure {output}
	smc_pad->Set_Parameters.MAX_POSITION = 0;
	smc_pad->Set_Parameters.MIN_POSITION = 0;
	smc_pad->Set_Parameters.MAX_VELOCITY = 0;
	smc_pad->Set_Parameters.MIN_POSITION = 0;
	smc_pad->Actual_Parameters.motorTemperature = 0;
	smc_pad->Actual_Parameters.position = 0;
	smc_pad->Actual_Parameters.torque = 0;
	smc_pad->Actual_Parameters.velocity = 0;
	// Other output parameters}
	smc_pad->Active = 0;
	smc_pad->Actual_State = 0;
	smc_pad->PowerOn = 0;
	smc_pad->Status = 0;
	smc_pad->InPosition = 0;
} // end function

// **************** PARAMETERS {NULL} **********************//
void parameters_null(struct SMC_PAD* smc_pad){
	// Parameters Mode structure {Input}
	smc_pad->Mode.home = 0;
	// Mode {automatic}
	smc_pad->Mode.automatic.instruction = INSTR_REAL_TIME;
	smc_pad->Mode.automatic.start       = 0;
	// Mode {manual}
	smc_pad->Mode.manual.start          = 0;
	// Set parameters structure {Input}
	smc_pad->Set_Parameters.position = 0;
	smc_pad->Set_Parameters.velocity = 0;
	// Set parameters {limit}
	smc_pad->Set_Parameters.limit.mode = INSTR_SIGNAL;
	smc_pad->Set_Parameters.limit.position_end   = 0;
	smc_pad->Set_Parameters.limit.position_start = 0;
	smc_pad->Set_Parameters.limit.signal         = 0;
	smc_pad->Set_Parameters.limit.time[0]        = 0;
	smc_pad->Set_Parameters.limit.time[1]        = 0;
	smc_pad->Set_Parameters.limit.velocity       = 0;
	// Signal {limit/in position}
	smc_pad->Set_Parameters.limit.signal_inPos[0] = 0;
	smc_pad->Set_Parameters.limit.signal_inPos[1] = 0;
	// Set parameters {sequence}
	smc_pad->Set_Parameters.sequence.mode = INSTR_SIGNAL;
	// Set parameters {sequence/position}
	smc_pad->Set_Parameters.sequence.position[0] = 0;
	smc_pad->Set_Parameters.sequence.position[1] = 0;
	smc_pad->Set_Parameters.sequence.position[2] = 0;
	smc_pad->Set_Parameters.sequence.position[3] = 0;
	smc_pad->Set_Parameters.sequence.position[4] = 0;
	// Set parameters {sequence/velocity}
	smc_pad->Set_Parameters.sequence.velocity[0] = 0;
	smc_pad->Set_Parameters.sequence.velocity[1] = 0;
	smc_pad->Set_Parameters.sequence.velocity[2] = 0;
	smc_pad->Set_Parameters.sequence.velocity[3] = 0;
	smc_pad->Set_Parameters.sequence.velocity[4] = 0;
	// Set parameters {sequence/time}
	smc_pad->Set_Parameters.sequence.time[0] = 0;
	smc_pad->Set_Parameters.sequence.time[1] = 0;
	smc_pad->Set_Parameters.sequence.time[2] = 0;
	smc_pad->Set_Parameters.sequence.time[3] = 0;
	smc_pad->Set_Parameters.sequence.time[4] = 0;
	// Signal {sequence/in position}
	smc_pad->Set_Parameters.sequence.signal_inPos[0] = 0;
	smc_pad->Set_Parameters.sequence.signal_inPos[1] = 0;
	smc_pad->Set_Parameters.sequence.signal_inPos[2] = 0;
	smc_pad->Set_Parameters.sequence.signal_inPos[3] = 0;
	smc_pad->Set_Parameters.sequence.signal_inPos[4] = 0;
} // end function

// **************** UPDATE CYCLIC PARAMETERS **********************//
void update_cyclicParameters(struct SMC_PAD* smc_pad, LREAL position, LREAL velocity){
	if(smc_pad->MpAxisCyclic->CyclicSetActive == 1){
		smc_pad->MpAxisCyclic->CyclicPosition = 0;
	}

	if(smc_pad->MpAxisCyclic->CyclicSetActive == 0){
		smc_pad->MpAxisCyclicParType->PositionModeMaxVelocity = (REAL)(velocity);
		smc_pad->MpAxisCyclicParType->Acceleration            = (REAL)(smc_pad->MpAxisCyclicParType->PositionModeMaxVelocity/(fabs(position)/velocity));
		smc_pad->MpAxisCyclicParType->Deceleration            = (REAL)(smc_pad->MpAxisCyclicParType->PositionModeMaxVelocity/(fabs(position)/velocity));
	}
} // end function

// **************** SET TIME **********************//
BOOL set_time(BOOL enable, TIME t){
	ton_1.IN = enable;
	ton_1.PT = t;

	TON(&ton_1);

	return ton_1.Q;
} // end function
```

### Data object Logical/Motion_Package/acp10etxen (Ett)

- acp10etxen.ett (not shown)

### Package Logical/Motion_Package/gAxis01_Xobj - gAxis01_Xobj

- Data object Logical/Motion_Package/gAxis01_Xobj/gAxis01_Xa (Apt) (no source held here)

### Data object Logical/Motion_Package/gAxis01_Xobj/gAxis01_Xi (Ax)

#### gAxis01_Xi.ax
```
InitParameter (Version=5.12.2, NcSwId=Acp10)
  ACP10AXIS_typ:
    dig_in:
      level:
        reference = ncACTIV_HI
        pos_hw_end = ncACTIV_HI
        neg_hw_end = ncACTIV_HI
        trigger1 = ncACTIV_HI
        trigger2 = ncACTIV_HI
    encoder_if:
      parameter:
        count_dir = ncSTANDARD
        scaling:
          load:
            units = 540
            rev_motor = 1
    limit:
      parameter:
        v_pos = 10000
        v_neg = 10000
        a1_pos = 50000
        a2_pos = 50000
        a1_neg = 50000
        a2_neg = 50000
        t_jolt = 0
        t_in_pos = 0
        pos_sw_end = 2000000000
        neg_sw_end = -2000000000
        ds_warning = 500
        ds_stop = 1000
        a_stop = 1.0e30
        dv_stop = 0
        dv_stop_mode = ncOFF
    controller:
      mode = ncPOSITION
      position:
        kv = 50
        tn = 0
        t_predict = 0.0004
        t_total = 0.0004
        p_max = 1.0e30
        i_max = 0
      speed:
        kv = 2.0
        tn = 0
        t_filter = 0.0
        isq_filter1:
          type = ncOFF
          a0 = 0.0
          a1 = 0.0
          b0 = 0.0
          b1 = 0.0
          b2 = 0.0
          c0_par_id = 0
          c1_par_id = 0
        isq_filter2:
          type = ncOFF
          a0 = 0.0
          a1 = 0.0
          b0 = 0.0
          b1 = 0.0
          b2 = 0.0
          c0_par_id = 0
          c1_par_id = 0
        isq_filter3:
          type = ncOFF
          a0 = 0.0
          a1 = 0.0
          b0 = 0.0
          b1 = 0.0
          b2 = 0.0
          c0_par_id = 0
          c1_par_id = 0
      uf:
        type = ncLINEAR + ncCORRECTION
        auto_config = ncMOTOR_PAR
        u0 = 0
        un = 0
        fn = 50.0
        k_f_slip = 0
      ff:
        mode = ncSTANDARD
        torque_load = 0.0
        torque_pos = 0.0
        torque_neg = 0.0
        kv_torque = 0.0
        inertia = 0.0
        t_filter_a = 0.0
      fb:
        mode = ncSTANDARD
        speed_mix_ratio = 0.0
        speed_kv = 2.0
      model:
        mass1:
          inertia = 0
          viscous_friction = 0
        mass2:
          inertia = 0
          viscous_friction = 0
          stiffness = 0
          damping = 0
    move:
      stop:
        parameter[0]:
          decel_ramp = ncA_LIMIT
          controller = ncON
        parameter[1]:
          decel_ramp = ncA_LIMIT
          controller = ncON
        parameter[2]:
          decel_ramp = ncA_LIMIT
          controller = ncON
        parameter[3]:
          decel_ramp = ncA_LIMIT
          controller = ncON
        quickstop:
          decel_ramp = ncA_LIMIT
          t_jolt = 0
        drive_error:
          decel_ramp = ncA_LIMIT
      homing:
        parameter:
          s = 0
          v_switch = 5000
          v_trigger = 500
          a = 50000
          mode = ncDIRECT
          edge_sw = ncPOSITIVE
          start_dir = ncPOSITIVE
          trigg_dir = ncPOSITIVE
          ref_pulse = ncOFF
          fix_dir = ncOFF
          tr_s_block = 0
          torque_lim = 0
          ds_block = 0
          ds_stop = 0
      basis:
        parameter:
          v_pos = 5000
          v_neg = 5000
          a1_pos = 50000
          a2_pos = 50000
          a1_neg = 50000
          a2_neg = 50000
    message:
      text:
        parameter:
          format = ncBREAK
          columns = 80
          data_modul = acp10etxen
```


- Data object Logical/Motion_Package/gAxis01_Yobj/gAxis01_Ya (Apt) (no source held here)

- Data object Logical/Motion_Package/gAxis01_Yobj/gAxis01_Yi (Ax) (no source held here)

### Package Logical/Motion_Package/gAxis01_Zobj - gAxis01_Zobj

- Data object Logical/Motion_Package/gAxis01_Zobj/gAxis01_Za (Apt) (no source held here)

### Data object Logical/Motion_Package/gAxis01_Zobj/gAxis01_Zi (Ax)

#### gAxis01_Zi.ax
```
InitParameter (Version=5.12.2, NcSwId=Acp10)
  ACP10AXIS_typ:
    dig_in:
      level:
        reference = ncACTIV_HI
        pos_hw_end = ncACTIV_LO
        neg_hw_end = ncACTIV_LO
        trigger1 = ncACTIV_HI
        trigger2 = ncACTIV_LO + ncQUICKSTOP
    encoder_if:
      parameter:
        count_dir = ncSTANDARD
        scaling:
          load:
            units = 540
            rev_motor = 1
    limit:
      parameter:
        v_pos = 10000
        v_neg = 10000
        a1_pos = 50000
        a2_pos = 50000
        a1_neg = 50000
        a2_neg = 50000
        t_jolt = 0
        t_in_pos = 0
        pos_sw_end = 2000000000
        neg_sw_end = -2000000000
        ds_warning = 500
        ds_stop = 1000
        a_stop = 1.0e30
        dv_stop = 0
        dv_stop_mode = ncOFF
    controller:
      mode = ncPOSITION
      position:
        kv = 50
        tn = 0
        t_predict = 0.0004
        t_total = 0.0004
        p_max = 1.0e30
        i_max = 0
      speed:
        kv = 2.0
        tn = 0
        t_filter = 0.0
        isq_filter1:
          type = ncOFF
          a0 = 0.0
          a1 = 0.0
          b0 = 0.0
          b1 = 0.0
          b2 = 0.0
          c0_par_id = 0
          c1_par_id = 0
        isq_filter2:
          type = ncOFF
          a0 = 0.0
          a1 = 0.0
          b0 = 0.0
          b1 = 0.0
          b2 = 0.0
          c0_par_id = 0
          c1_par_id = 0
        isq_filter3:
          type = ncOFF
          a0 = 0.0
          a1 = 0.0
          b0 = 0.0
          b1 = 0.0
          b2 = 0.0
          c0_par_id = 0
          c1_par_id = 0
      uf:
        type = ncLINEAR + ncCORRECTION
        auto_config = ncMOTOR_PAR
        u0 = 0
        un = 0
        fn = 50.0
        k_f_slip = 0
      ff:
        mode = ncSTANDARD
        torque_load = 0.0
        torque_pos = 0.0
        torque_neg = 0.0
        kv_torque = 0.0
        inertia = 0.0
        t_filter_a = 0.0
      fb:
        mode = ncSTANDARD
        speed_mix_ratio = 0.0
        speed_kv = 2.0
      model:
        mass1:
          inertia = 0
          viscous_friction = 0
        mass2:
          inertia = 0
          viscous_friction = 0
          stiffness = 0
          damping = 0
    move:
      stop:
        parameter[0]:
          decel_ramp = ncA_LIMIT
          controller = ncON
        parameter[1]:
          decel_ramp = ncA_LIMIT
          controller = ncON
        parameter[2]:
          decel_ramp = ncA_LIMIT
          controller = ncON
        parameter[3]:
          decel_ramp = ncA_LIMIT
          controller = ncON
        quickstop:
          decel_ramp = ncA_LIMIT
          t_jolt = 0
        drive_error:
          decel_ramp = ncA_LIMIT
      homing:
        parameter:
          s = 0
          v_switch = 5000
          v_trigger = 500
          a = 50000
          mode = ncDIRECT
          edge_sw = ncPOSITIVE
          start_dir = ncPOSITIVE
          trigg_dir = ncPOSITIVE
          ref_pulse = ncOFF
          fix_dir = ncOFF
          tr_s_block = 0
          torque_lim = 0
          ds_block = 0
          ds_stop = 0
      basis:
        parameter:
          v_pos = 5000
          v_neg = 5000
          a1_pos = 50000
          a2_pos = 50000
          a1_neg = 50000
          a2_neg = 50000
    message:
      text:
        parameter:
          format = ncBREAK
          columns = 80
          data_modul = acp10etxen
```

### Package Logical/Motion_Package/gAxis01_Cobj - gAxis01_Cobj

### Data object Logical/Motion_Package/gAxis01_Cobj/gAxis01_Ca (Apt)

#### gAxis01_Ca.apt
```
AcoposParameterTable:
  Root Parameters
```

- Data object Logical/Motion_Package/gAxis01_Cobj/gAxis01_Ci (Ax) (no source held here)

### Program Logical/Main_Control/Main (ANSIC)

#### Main.c
```c
/**
 * MIT License
 * Copyright(c) 2020 Roman Parak
 * Permission is hereby granted, free of charge, to any person obtaining a copy
 * of this software and associated documentation files (the "Software"), to deal
 * in the Software without restriction, including without limitation the rights
 * to use, copy, modify, merge, publish, distribute, sublicense, and/or sell
 * copies of the Software, and to permit persons to whom the Software is
 * furnished to do so, subject to the following conditions:
 * The above copyright notice and this permission notice shall be included in all
 * copies or substantial portions of the Software.
 * THE SOFTWARE IS PROVIDED "AS IS", WITHOUT WARRANTY OF ANY KIND, EXPRESS OR
 * IMPLIED, INCLUDING BUT NOT LIMITED TO THE WARRANTIES OF MERCHANTABILITY,
 * FITNESS FOR A PARTICULAR PURPOSE AND NONINFRINGEMENT. IN NO EVENT SHALL THE
 * AUTHORS OR COPYRIGHT HOLDERS BE LIABLE FOR ANY CLAIM, DAMAGES OR OTHER
 * LIABILITY, WHETHER IN AN ACTION OF CONTRACT, TORT OR OTHERWISE, ARISING FROM,
 * OUT OF OR IN CONNECTION WITH THE SOFTWARE OR THE USE OR OTHER DEALINGS IN THE
 * SOFTWARE.
 */
/**
 * Author   : Roman Parak
 * Email    : Roman.Parak@outlook.com
 * File Name: Main.c
 */

#include <bur/plctypes.h>
#include <standard.h>

#ifdef _DEFAULT_INCLUDES
#include <AsDefault.h>
#endif

// Time Function Block
_LOCAL TON_typ ton_1;
// Output Variable
_LOCAL BOOL wait_var;
// Time in ms
_LOCAL TIME wait_time;
// Auxliliary variables (Counter)
_LOCAL USINT aux_counter_main_sm_act, aux_counter_main_sm_bef;
_LOCAL USINT aux_counter_brP_sm_act, aux_counter_brP_sm_bef;
_LOCAL USINT aux_counter_smcP_sm_act, aux_counter_smcP_sm_bef;
// Offset Variables
// Initialization Pad (Start Positon)
_LOCAL LREAL offset_init_pad_x[9];
_LOCAL LREAL offset_init_pad_y[9];
// BR Pad (End Position Warehouse)
_LOCAL LREAL offset_br_pad_x[4];
_LOCAL LREAL offset_br_pad_y[4];
// SMC Pad (End Position Warehouse)
_LOCAL LREAL offset_smc_pad_x[4];
_LOCAL LREAL offset_smc_pad_y[4];

// FUNCTION // DECLARATION //
BOOL set_time(BOOL enable, TIME t);

// OBJECT TYPE
const BOOL OBJ_TYPE_BR  = 2;
const BOOL OBJ_TYPE_SMC = 1;
const BOOL OBJ_TYPE_ERR = 10;
// XYZ MANIPULATOR
const LREAL INIT_PAD_OFFSET_X  = 345.0;
const LREAL INIT_PAD_OFFSET_Y  = 660.0;
const LREAL INIT_PAD_OFFSET_Z  = 1255.0;
const LREAL INIT_CC_OFFSET_X   = 6425.0;
const LREAL INIT_CC_OFFSET_Y   = 2960.0;
const LREAL INIT_CC_OFFSET_Z   = 1072.0;
const LREAL INIT_BRW_OFFSET_X  = 2895.0;
const LREAL INIT_BRW_OFFSET_Y  = 4060.0;
const LREAL INIT_BRW_OFFSET_Z  = 1255.0;
const LREAL INIT_SMCW_OFFSET_X = 395.0;
const LREAL INIT_SMCW_OFFSET_Y = 4060.0;
const LREAL INIT_SMCW_OFFSET_Z = 1255.0;
// CAMEA CONVEYOR
const LREAL INIT_CC_MAIN_OFFSET_X = 3500;
// BOTH
const LREAL HOME_POS = 0.0;

void _INIT ProgramInit(void)
{
	// -------------------- INITIALIZATION Digita-Twin Main Global Variable -------------------- //
	// Camera Scanning Variable
	dT_Main.camera.scan = 0;
	// Actual Position of the XYZ Manipulator and Camera Conveyor (Read from task X_AXIS_M, etc.)
	dT_Main.camera_conveyor.X.actual_position = 0;
	dT_Main.xyz_manipulator.X.actual_position = 0;
	dT_Main.xyz_manipulator.Y.actual_position = 0;
	dT_Main.xyz_manipulator.Z.actual_position = 0;
	// Mani Control State Variable
	dT_Main.service.actual_state = 0;
	// Object Control (Read / Write Variable)
	dT_Main.service.object.write.attach        = 0;
	dT_Main.service.object.write.detach        = 0;
	dT_Main.service.object.write.reset         = 0;
	dT_Main.service.object.write.set_object_id = 0;
	dT_Main.service.object.read.object_id   = 0;
	dT_Main.service.object.read.object_type = 0;
	// Initial Parameters (Velocity, Start State)
	dT_Main.xyz_manipulator.X.parameter.vel = 3500;
	dT_Main.xyz_manipulator.X.actual_state  = LINP_CTRL_WAIT_STATE;
	dT_Main.xyz_manipulator.Y.parameter.vel = 2500;
	dT_Main.xyz_manipulator.Y.actual_state  = LINP_CTRL_WAIT_STATE;
	dT_Main.xyz_manipulator.Z.parameter.vel = 2000;
	dT_Main.xyz_manipulator.Z.actual_state  = LINP_CTRL_WAIT_STATE;
	dT_Main.camera_conveyor.X.parameter.vel = 2500;
	dT_Main.camera_conveyor.X.actual_state  = LINP_CTRL_WAIT_STATE;

	// -------------------- INITIALIZATION Offset Parameter for the Motion -------------------- //
	// Initialization Pad (Start Positon)
	offset_init_pad_x[0] = 0.0; offset_init_pad_y[0]    = 0.0;
	offset_init_pad_x[1] = 0.0; offset_init_pad_y[1]    = 800.0;
	offset_init_pad_x[2] = 0.0; offset_init_pad_y[2]    = 1600.0;
	offset_init_pad_x[3] = 600.0; offset_init_pad_y[3]  = 0.0;
	offset_init_pad_x[4] = 600.0; offset_init_pad_y[4]  = 800.0;
	offset_init_pad_x[5] = 600.0; offset_init_pad_y[5]  = 1600.0;
	offset_init_pad_x[6] = 1200.0; offset_init_pad_y[6] = 0.0;
	offset_init_pad_x[7] = 1200.0; offset_init_pad_y[7] = 800.0;
	offset_init_pad_x[8] = 1200.0; offset_init_pad_y[8] = 1600.0;
	// BR Pad (End Position Warehouse)
	offset_br_pad_x[0] = 0.0; offset_br_pad_y[0]   = 0.0;
	offset_br_pad_x[1] = 0.0; offset_br_pad_y[1]   = 800.0;
	offset_br_pad_x[2] = 600.0; offset_br_pad_y[2] = 0.0;
	offset_br_pad_x[3] = 600.0; offset_br_pad_y[3] = 800.0;
	// SMC Pad (End Position Warehouse)
	offset_smc_pad_x[0] = 0.0; offset_smc_pad_y[0]   = 0.0;
	offset_smc_pad_x[1] = 0.0; offset_smc_pad_y[1]   = 800.0;
	offset_smc_pad_x[2] = 600.0; offset_smc_pad_y[2] = 0.0;
	offset_smc_pad_x[3] = 600.0; offset_smc_pad_y[3] = 800.0;

	// Wait 1 second at a certain step
	wait_time = 1000;

	// Reset Counters
	aux_counter_main_sm_act = aux_counter_main_sm_bef = 0;
	aux_counter_brP_sm_act  = aux_counter_brP_sm_bef  = 0;
	aux_counter_smcP_sm_act = aux_counter_smcP_sm_bef = 0;

}

void _CYCLIC ProgramCyclic(void)
{
	switch(dT_Main.service.actual_state){
		case 0: // INITIALIZATION STAT
			{
				if(dT_Main.camera_conveyor.X.active == 1 && dT_Main.xyz_manipulator.X.active == 1 && dT_Main.xyz_manipulator.Y.active == 1 && dT_Main.xyz_manipulator.Z.active == 1){
					dT_Main.service.mapp_view.active = 1;
					dT_Main.service.actual_state = 1;
				}
			}
			break;

		case 1: // POWER STATE
			{
				if(dT_Main.service.power == 1){
					if(dT_Main.camera_conveyor.X.power_on == 1 && dT_Main.xyz_manipulator.X.power_on == 1 && dT_Main.xyz_manipulator.Y.power_on == 1 && dT_Main.xyz_manipulator.Z.power_on == 1){
						dT_Main.service.mapp_view.power_on = 1;
						dT_Main.service.actual_state = 2;
					}
				}
			}
			break;

		case 2: // HOME STATE
			{
				if(dT_Main.service.home == 1){
					if(dT_Main.camera_conveyor.X.is_homed == 1 && dT_Main.xyz_manipulator.X.is_homed == 1 && dT_Main.xyz_manipulator.Y.is_homed == 1 && dT_Main.xyz_manipulator.Z.is_homed == 1){
						dT_Main.service.mapp_view.is_homed = 1;
						dT_Main.service.actual_state = 3;
					}
				}
			}
			break;

		case 3: // START STATE
			{
				if(dT_Main.service.start == 1){
					dT_Main.camera_conveyor.X.start = 1;
					dT_Main.xyz_manipulator.X.start = 1;
					dT_Main.xyz_manipulator.Y.start = 1;
					dT_Main.xyz_manipulator.Z.start = 1;
					dT_Main.service.actual_state = 4;
				}
			}
			break;

		case 4: // MOVE INIT POS (1) -> OBJECT_{i} DETACHED
			{
				aux_counter_main_sm_bef = aux_counter_main_sm_act;
				aux_counter_brP_sm_bef  = aux_counter_brP_sm_act;
				aux_counter_smcP_sm_bef = aux_counter_smcP_sm_act;

				dT_Main.service.start = 0;

				dT_Main.xyz_manipulator.X.parameter.pos = INIT_PAD_OFFSET_X + offset_init_pad_x[dT_Main.service.object.read.object_id];
				dT_Main.xyz_manipulator.Y.parameter.pos = INIT_PAD_OFFSET_Y + offset_init_pad_y[dT_Main.service.object.read.object_id];
				dT_Main.xyz_manipulator.Z.parameter.pos = HOME_POS;
				dT_Main.camera_conveyor.X.parameter.pos = HOME_POS;

				if((dT_Main.xyz_manipulator.X.actual_position == dT_Main.xyz_manipulator.X.parameter.pos) && (dT_Main.xyz_manipulator.Y.actual_position == dT_Main.xyz_manipulator.Y.parameter.pos) && (dT_Main.xyz_manipulator.Z.actual_position == dT_Main.xyz_manipulator.Z.parameter.pos)
				&& (dT_Main.camera_conveyor.X.actual_position == dT_Main.camera_conveyor.X.parameter.pos)){
					dT_Main.service.actual_state = 5;
				}

			}
			break;

		case 5: // MOVE INIT POS (2) -> OBJECT_{i} DETACHED
			{
				dT_Main.xyz_manipulator.Z.parameter.pos = INIT_PAD_OFFSET_Z;

				if(dT_Main.xyz_manipulator.Z.actual_position == dT_Main.xyz_manipulator.Z.parameter.pos){
					dT_Main.service.actual_state = 6;
				}

			}
			break;

		case 6: // MOVE INIT POS (3) -> OBJECT_{i} ATTACHED (Wait 1s)
			{
				dT_Main.service.object.write.attach = 1;
				wait_var = set_time(1, wait_time);

				if(wait_var == 1){
					dT_Main.service.actual_state = 7;
					dT_Main.service.object.write.attach = 0;
					wait_var = set_time(0, wait_time);
				}
			}
			break;

		case 7: // MOVE INIT POS (4) -> OBJECT_{i} ATTACHED
			{
				dT_Main.xyz_manipulator.Z.parameter.pos = HOME_POS;

				if(dT_Main.xyz_manipulator.Z.actual_position == dT_Main.xyz_manipulator.Z.parameter.pos){
					dT_Main.service.actual_state = 8;
				}
			}
			break;

		case 8: // MOVE CAMERA CONVEYOR POS (1) -> OBJECT_{i} ATTACHED
			{
				dT_Main.xyz_manipulator.X.parameter.pos = INIT_CC_OFFSET_X;
				dT_Main.xyz_manipulator.Y.parameter.pos = INIT_CC_OFFSET_Y;

				if((dT_Main.xyz_manipulator.X.actual_position == dT_Main.xyz_manipulator.X.parameter.pos) && (dT_Main.xyz_manipulator.Y.actual_position == dT_Main.xyz_manipulator.Y.parameter.pos)){
					dT_Main.service.actual_state = 9;
				}
			}
			break;

		case 9: // MOVE CAMERA CONVEYOR POS (2) -> OBJECT_{i} ATTACHED
			{
				dT_Main.xyz_manipulator.Z.parameter.pos = INIT_CC_OFFSET_Z;

				if(dT_Main.xyz_manipulator.Z.actual_position == dT_Main.xyz_manipulator.Z.parameter.pos){
					dT_Main.service.actual_state = 10;
				}
			}
			break;

		case 10: // MOVE CAMERA CONVEYOR POS (3) -> OBJECT_{i} DETACHED XYZ and ATTACHED CAMERA CONVEYOR
			{
				dT_Main.service.object.write.detach = 1;
				wait_var     = set_time(1, wait_time);

				if(wait_var == 1){
					dT_Main.service.actual_state = 11;
					dT_Main.service.object.write.detach = 0;
					wait_var     = set_time(0, wait_time);
				}
			}
			break;

		case 11: // MOVE CAMERA CONVEYOR POS (4) -> OBJECT_{i} DETACHED XYZ and ATTACHED CAMERA CONVEYOR
			{
				dT_Main.xyz_manipulator.Z.parameter.pos = HOME_POS;
				dT_Main.camera_conveyor.X.parameter.pos = INIT_CC_MAIN_OFFSET_X;

				if((dT_Main.xyz_manipulator.Z.actual_position == dT_Main.xyz_manipulator.Z.parameter.pos) && (dT_Main.camera_conveyor.X.actual_position == dT_Main.camera_conveyor.X.parameter.pos)){
					dT_Main.service.actual_state = 12;
				}
			}
			break;

		case 12: // MOVE CAMERA CONVEYOR POS (5) -> OBJECT_{i} DETACHED XYZ and ATTACHED CAMERA CONVEYOR (Wait 0.5s)
			{
				dT_Main.camera.scan          = 1;
				wait_var     = set_time(1, wait_time / 2);

				if(wait_var == 1){
					dT_Main.service.actual_state = 13;
					dT_Main.camera.scan          = 0;
					wait_var     = set_time(0, wait_time);
				}
			}
			break;

		case 13: // MOVE CAMERA CONVEYOR POS (6) -> OBJECT_{i} DETACHED XYZ and ATTACHED CAMERA CONVEYOR
			{
				dT_Main.xyz_manipulator.Z.parameter.pos = HOME_POS;
				dT_Main.camera_conveyor.X.parameter.pos = HOME_POS;

				if((dT_Main.xyz_manipulator.Z.actual_position == dT_Main.xyz_manipulator.Z.parameter.pos) && (dT_Main.camera_conveyor.X.actual_position == dT_Main.camera_conveyor.X.parameter.pos)){
					dT_Main.service.actual_state = 14;
				}
			}
			break;

		case 14: // MOVE CAMERA CONVEYOR POS (7) -> OBJECT_{i} ATTACHED XYZ and DETACHED CAMERA CONVEYOR
			{
				dT_Main.xyz_manipulator.Z.parameter.pos = INIT_CC_OFFSET_Z;

				if(dT_Main.xyz_manipulator.Z.actual_position == dT_Main.xyz_manipulator.Z.parameter.pos){
					dT_Main.service.actual_state = 15;
				}
			}
			break;

		case 15: // MOVE CAMERA CONVEYOR POS (8) -> OBJECT_{i} ATTACHED XYZ and DETACHED CAMERA CONVEYOR (Wait 1s)
			{
				dT_Main.service.object.write.attach = 1;
				wait_var     = set_time(1, wait_time);

				if(wait_var == 1){
					dT_Main.service.actual_state = 16;
					dT_Main.service.object.write.attach = 0;
					wait_var     = set_time(0, wait_time);
				}
			}
			break;

		case 16: // MOVE CAMERA CONVEYOR POS (9) -> OBJECT_{i} ATTACHED XYZ and DETACHED CAMERA CONVEYOR
			{
				dT_Main.xyz_manipulator.Z.parameter.pos = HOME_POS;

				if(dT_Main.xyz_manipulator.Z.actual_position == dT_Main.xyz_manipulator.Z.parameter.pos){
					dT_Main.service.actual_state = 17;
				}
			}
			break;

		case 17: // WAIT STATE -> GET THE OBJECT TYPE
			{
				if(dT_Main.service.object.read.object_type == OBJ_TYPE_ERR){
					dT_Main.service.actual_state = 20;
				}else if(dT_Main.service.object.read.object_type == OBJ_TYPE_BR){
					dT_Main.service.actual_state = 30;
				}else if(dT_Main.service.object.read.object_type == OBJ_TYPE_SMC){
					dT_Main.service.actual_state = 40;
				}
			}
			break;

		case 20: // TRASH STATE (1) -> OBJECT_{i} ATTACHED XYZ
			{
				dT_Main.xyz_manipulator.X.parameter.pos = 3500.0;
				dT_Main.xyz_manipulator.Y.parameter.pos = 1750.0;

				if((dT_Main.xyz_manipulator.X.actual_position == dT_Main.xyz_manipulator.X.parameter.pos) && (dT_Main.xyz_manipulator.Y.actual_position == dT_Main.xyz_manipulator.Y.parameter.pos)){
					dT_Main.service.actual_state = 21;
				}
			}
			break;

		case 21: // TRASH STATE (2) -> OBJECT_{i} ATTACHED XYZ
			{
				dT_Main.xyz_manipulator.Z.parameter.pos = 1000.0;

				if(dT_Main.xyz_manipulator.Z.actual_position == dT_Main.xyz_manipulator.Z.parameter.pos){
					dT_Main.service.actual_state = 22;
				}
			}
			break;

		case 22: // TRASH STATE (3) -> OBJECT_{i} DETACHED XYZ (Wait 1s)
			{
				dT_Main.service.object.write.detach = 1;
				wait_var     = set_time(1, wait_time);

				if(wait_var == 1){
					dT_Main.service.actual_state = 23;
					dT_Main.service.object.write.detach = 0;
					wait_var     = set_time(0, wait_time);
				}
			}
			break;

		case 23: // TRASH STATE (4) -> OBJECT_{i} is in the Trash
			{
				dT_Main.xyz_manipulator.Z.parameter.pos = HOME_POS;

				if(dT_Main.xyz_manipulator.Z.actual_position == dT_Main.xyz_manipulator.Z.parameter.pos){
					dT_Main.service.actual_state = 50;
				}
			}
			break;

		case 30: // BR WAREHOUSE STATE (1) -> OBJECT_{i} ATTACHED XYZ
			{
				dT_Main.xyz_manipulator.X.parameter.pos = INIT_BRW_OFFSET_X + offset_br_pad_x[aux_counter_brP_sm_act];
				dT_Main.xyz_manipulator.Y.parameter.pos = INIT_BRW_OFFSET_Y + offset_br_pad_y[aux_counter_brP_sm_act];

				if((dT_Main.xyz_manipulator.X.actual_position == dT_Main.xyz_manipulator.X.parameter.pos) && (dT_Main.xyz_manipulator.Y.actual_position == dT_Main.xyz_manipulator.Y.parameter.pos)){
					dT_Main.service.actual_state = 31;
				}
			}
			break;

		case 31: // BR WAREHOUSE STATE (2) -> OBJECT_{i} ATTACHED XYZ
			{
				dT_Main.xyz_manipulator.Z.parameter.pos = INIT_BRW_OFFSET_Z;

				if(dT_Main.xyz_manipulator.Z.actual_position == dT_Main.xyz_manipulator.Z.parameter.pos){
					dT_Main.service.actual_state = 32;
				}
			}
			break;

		case 32: // BR WAREHOUSE STATE (3) -> OBJECT_{i} DETACHED XYZ (Wait 1s)
			{
				dT_Main.service.object.write.detach = 1;
				wait_var     = set_time(1, wait_time);

				if(wait_var == 1){
					dT_Main.service.actual_state = 33;
					dT_Main.service.object.write.detach = 0;
					wait_var     = set_time(0, wait_time);
				}
			}
			break;

		case 33: // BR WAREHOUSE STATE (4) -> OBJECT_{i} is in the BR WAREHOUSE
			{
				dT_Main.xyz_manipulator.Z.parameter.pos = HOME_POS;

				if(dT_Main.xyz_manipulator.Z.actual_position == dT_Main.xyz_manipulator.Z.parameter.pos){
					if(aux_counter_brP_sm_act == aux_counter_brP_sm_bef){
						aux_counter_brP_sm_act = aux_counter_brP_sm_bef + 1;
					}

					dT_Main.service.actual_state = 50;
				}
			}
			break;

		case 40: // SMC WAREHOUSE STATE (1) -> OBJECT_{i} ATTACHED XYZ
			{
				dT_Main.xyz_manipulator.X.parameter.pos = INIT_SMCW_OFFSET_X + offset_smc_pad_x[aux_counter_smcP_sm_act];
				dT_Main.xyz_manipulator.Y.parameter.pos = INIT_SMCW_OFFSET_Y + offset_smc_pad_y[aux_counter_smcP_sm_act];

				if((dT_Main.xyz_manipulator.X.actual_position == dT_Main.xyz_manipulator.X.parameter.pos) && (dT_Main.xyz_manipulator.Y.actual_position == dT_Main.xyz_manipulator.Y.parameter.pos)){
					dT_Main.service.actual_state = 41;
				}
			}
			break;

		case 41: // SMC WAREHOUSE STATE (1) -> OBJECT_{i} ATTACHED XYZ
			{
				dT_Main.xyz_manipulator.Z.parameter.pos = INIT_SMCW_OFFSET_Z;

				if(dT_Main.xyz_manipulator.Z.actual_position == dT_Main.xyz_manipulator.Z.parameter.pos){
					dT_Main.service.actual_state = 42;
				}
			}
			break;

		case 42: // SMC WAREHOUSE STATE (3) -> OBJECT_{i} DETACHED XYZ (Wait 1s)
			{
				dT_Main.service.object.write.detach = 1;
				wait_var     = set_time(1, wait_time);

				if(wait_var == 1){
					dT_Main.service.actual_state = 43;
					dT_Main.service.object.write.detach = 0;
					wait_var     = set_time(0, wait_time);
				}
			}
			break;

		case 43: // SMC WAREHOUSE STATE (4) -> OBJECT_{i} is in the SMC WAREHOUSE
			{
				dT_Main.xyz_manipulator.Z.parameter.pos = HOME_POS;

				if(dT_Main.xyz_manipulator.Z.actual_position == dT_Main.xyz_manipulator.Z.parameter.pos){

					if(aux_counter_smcP_sm_act == aux_counter_smcP_sm_bef){
						aux_counter_smcP_sm_act = aux_counter_smcP_sm_bef + 1;
					}

					dT_Main.service.actual_state = 50;
				}
			}
			break;

		case 50: // MOVE INITIALIZATION POS (1) -> COUNTER +1
			{
				if(aux_counter_main_sm_act == aux_counter_main_sm_bef){
					aux_counter_main_sm_act = aux_counter_main_sm_bef + 1;
				}

				if(aux_counter_main_sm_act != 9){
					dT_Main.service.actual_state = 51;
				}else{
					dT_Main.service.actual_state = 60;
				}
			}
			break;

		case 51: // MOVE INITIALIZATION POS (2) -> (Wait 0.5s)
			{
				dT_Main.service.object.write.set_object_id = aux_counter_main_sm_act;
				wait_var     = set_time(1, wait_time/2);

				if(wait_var == 1){
					dT_Main.service.actual_state = 4;
					wait_var     = set_time(0, wait_time);
				}
			}
			break;

		case 60: // MOVE INITIALIZATION POS (3) -> Reset Variables
			{
				aux_counter_main_sm_act = aux_counter_main_sm_bef = 0;
				aux_counter_brP_sm_act  = aux_counter_brP_sm_bef  = 0;
				aux_counter_smcP_sm_act = aux_counter_smcP_sm_bef = 0;

				dT_Main.service.object.write.set_object_id = 0;

				dT_Main.xyz_manipulator.X.parameter.pos = INIT_PAD_OFFSET_X + offset_init_pad_x[0];
				dT_Main.xyz_manipulator.Y.parameter.pos = INIT_PAD_OFFSET_Y + offset_init_pad_y[0];

				if((dT_Main.xyz_manipulator.X.actual_position == dT_Main.xyz_manipulator.X.parameter.pos) && (dT_Main.xyz_manipulator.Y.actual_position == dT_Main.xyz_manipulator.Y.parameter.pos)){
					dT_Main.service.actual_state = 61;
				}
			}
			break;

		case 61: // WAIT STATE -> Wait for the user to reset the startup command
			{
				if(dT_Main.service.start == 1){
					dT_Main.service.actual_state = 4;
				}
			}
			break;

	}

	// **************** MappView -> Display the scanned object ********************** //
	if(dT_Main.service.object.read.object_type == OBJ_TYPE_ERR){
		dT_Main.service.mapp_view.cam_obj_id = 3;
	}else if(dT_Main.service.object.read.object_type == OBJ_TYPE_BR){
		dT_Main.service.mapp_view.cam_obj_id = 1;
	}else if(dT_Main.service.object.read.object_type == OBJ_TYPE_SMC){
		dT_Main.service.mapp_view.cam_obj_id = 2;
	}else{
		dT_Main.service.mapp_view.cam_obj_id = 0;
	}

	// **************** MappView -> Set the position of the object in the warehouse ********************** //
	if(aux_counter_brP_sm_act == 1){
		dT_Main.service.mapp_view.br_pad_obj_id[0] = 1;
		dT_Main.service.mapp_view.br_pad_obj_id[1] = 0;
		dT_Main.service.mapp_view.br_pad_obj_id[2] = 0;
		dT_Main.service.mapp_view.br_pad_obj_id[3] = 0;
	}else if(aux_counter_brP_sm_act == 2){
		dT_Main.service.mapp_view.br_pad_obj_id[0] = 1;
		dT_Main.service.mapp_view.br_pad_obj_id[1] = 1;
		dT_Main.service.mapp_view.br_pad_obj_id[2] = 0;
		dT_Main.service.mapp_view.br_pad_obj_id[3] = 0;
	}else if(aux_counter_brP_sm_act == 3){
		dT_Main.service.mapp_view.br_pad_obj_id[0] = 1;
		dT_Main.service.mapp_view.br_pad_obj_id[1] = 1;
		dT_Main.service.mapp_view.br_pad_obj_id[2] = 1;
		dT_Main.service.mapp_view.br_pad_obj_id[3] = 0;
	}else if(aux_counter_brP_sm_act == 4){
		dT_Main.service.mapp_view.br_pad_obj_id[0] = 1;
		dT_Main.service.mapp_view.br_pad_obj_id[1] = 1;
		dT_Main.service.mapp_view.br_pad_obj_id[2] = 1;
		dT_Main.service.mapp_view.br_pad_obj_id[3] = 1;
	}
	if(aux_counter_smcP_sm_act == 1){
		dT_Main.service.mapp_view.smc_pad_obj_id[0] = 1;
		dT_Main.service.mapp_view.smc_pad_obj_id[1] = 0;
		dT_Main.service.mapp_view.smc_pad_obj_id[2] = 0;
		dT_Main.service.mapp_view.smc_pad_obj_id[3] = 0;
	}else if(aux_counter_smcP_sm_act == 2){
		dT_Main.service.mapp_view.smc_pad_obj_id[0] = 1;
		dT_Main.service.mapp_view.smc_pad_obj_id[1] = 1;
		dT_Main.service.mapp_view.smc_pad_obj_id[2] = 0;
		dT_Main.service.mapp_view.smc_pad_obj_id[3] = 0;
	}else if(aux_counter_smcP_sm_act == 3){
		dT_Main.service.mapp_view.smc_pad_obj_id[0] = 1;
		dT_Main.service.mapp_view.smc_pad_obj_id[1] = 1;
		dT_Main.service.mapp_view.smc_pad_obj_id[2] = 1;
		dT_Main.service.mapp_view.smc_pad_obj_id[3] = 0;
	}else if(aux_counter_smcP_sm_act == 4){
		dT_Main.service.mapp_view.smc_pad_obj_id[0] = 1;
		dT_Main.service.mapp_view.smc_pad_obj_id[1] = 1;
		dT_Main.service.mapp_view.smc_pad_obj_id[2] = 1;
		dT_Main.service.mapp_view.smc_pad_obj_id[3] = 1;
	}

	// **************** MappView -> Reset ********************** //
	if(dT_Main.service.object.write.reset == 1){
		dT_Main.service.mapp_view.br_pad_obj_id[0] = 0;
		dT_Main.service.mapp_view.br_pad_obj_id[1] = 0;
		dT_Main.service.mapp_view.br_pad_obj_id[2] = 0;
		dT_Main.service.mapp_view.br_pad_obj_id[3] = 0;
		dT_Main.service.mapp_view.smc_pad_obj_id[0] = 0;
		dT_Main.service.mapp_view.smc_pad_obj_id[1] = 0;
		dT_Main.service.mapp_view.smc_pad_obj_id[2] = 0;
		dT_Main.service.mapp_view.smc_pad_obj_id[3] = 0;
	}
}

// **************** SET TIME **********************//
BOOL set_time(BOOL enable, TIME t){
	ton_1.IN = enable;
	ton_1.PT = t;

	TON(&ton_1);

	return ton_1.Q;
} // end function
```

### Program Logical/XYZ_MANIPULATOR/X_AXIS_M (ANSIC)

#### Main.c - Init, cyclic, exit code
```c
/**
 * MIT License
 * Copyright(c) 2020 Roman Parak
 * Permission is hereby granted, free of charge, to any person obtaining a copy
 * of this software and associated documentation files (the "Software"), to deal
 * in the Software without restriction, including without limitation the rights
 * to use, copy, modify, merge, publish, distribute, sublicense, and/or sell
 * copies of the Software, and to permit persons to whom the Software is
 * furnished to do so, subject to the following conditions:
 * The above copyright notice and this permission notice shall be included in all
 * copies or substantial portions of the Software.
 * THE SOFTWARE IS PROVIDED "AS IS", WITHOUT WARRANTY OF ANY KIND, EXPRESS OR
 * IMPLIED, INCLUDING BUT NOT LIMITED TO THE WARRANTIES OF MERCHANTABILITY,
 * FITNESS FOR A PARTICULAR PURPOSE AND NONINFRINGEMENT. IN NO EVENT SHALL THE
 * AUTHORS OR COPYRIGHT HOLDERS BE LIABLE FOR ANY CLAIM, DAMAGES OR OTHER
 * LIABILITY, WHETHER IN AN ACTION OF CONTRACT, TORT OR OTHERWISE, ARISING FROM,
 * OUT OF OR IN CONNECTION WITH THE SOFTWARE OR THE USE OR OTHER DEALINGS IN THE
 * SOFTWARE.
 */
/**
 * Author   : Roman Parak
 * Email    : Roman.Parak@outlook.com
 * File Name: Main.c
 */

#include <bur/plc.h>
#include <bur/plctypes.h>
#include "rp_funcx.h"

#ifdef _DEFAULT_INCLUDES
#include <AsDefault.h>
#endif

// {DEFINE - ABSOLUTE POSITION (Camera Conveyor AXIS}
#define Axis_XM_HOME_ABSOLUTE_POS 17700410;
// Camera Conveyor AXIS// MpAxis // STRUCT //
// {Camera Conveyor AXIS}
_LOCAL struct MpAxisBasic MpAxisBasic_Axis_XM;
_LOCAL struct MpAxisBasicParType MpAxis_Axis_XM_ParType;
// {Camera Conveyor AXIS}
_LOCAL struct MpAxisCyclicSet MpAxisCyclicSet_Axis_XM;
_LOCAL struct MpAxisCyclicSetParType AxisCyclicPar_Axis_XM;
// Camera Conveyor AXIS // SMC_PAD // STRUCT //
_LOCAL struct SMC_PAD Axis_XM_SMC_PAD;

void _INIT ProgramInit(void)
{
	// -------------------- INITIALIZATION MAPP AXIS -------------------- //
	// MpAxis SMC PAD //
	MpAxisBasic_Axis_XM.Enable         = 1;
	MpAxisBasic_Axis_XM.Axis           = &gAxis01_X;
	MpAxisBasic_Axis_XM.MpLink         = &gAxisBasic_Axis_M_X;
	MpAxisBasic_Axis_XM.Parameters     = &MpAxis_Axis_XM_ParType;
	// Cyclic Parameters {Read}
	MpAxis_Axis_XM_ParType.CyclicRead.MotorTempMode = mpAXIS_READ_CYCLIC;
	MpAxis_Axis_XM_ParType.CyclicRead.LagErrorMode  = mpAXIS_READ_CYCLIC;
	MpAxis_Axis_XM_ParType.CyclicRead.TorqueMode 	= mpAXIS_READ_CYCLIC;
	// MpAxisCyclicSet SMC PAD //
	MpAxisCyclicSet_Axis_XM.Enable 	= 1;
	MpAxisCyclicSet_Axis_XM.MpLink 	= &gAxisBasic_Axis_M_X;
	MpAxisCyclicSet_Axis_XM.Parameters = &AxisCyclicPar_Axis_XM;
	// MpAxisCyclicSet Parameters (initial) SMC PAD //
	AxisCyclicPar_Axis_XM.Acceleration            = 5000;
	AxisCyclicPar_Axis_XM.Deceleration            = 5000;
	AxisCyclicPar_Axis_XM.PositionModeMaxVelocity = 5000;

	// -------------------- INITIALIZATION SMCTrak -------------------- //
	// Camera Conveyor //
	// MpAxis & MpAxis Cyclic declaration
	Axis_XM_SMC_PAD.MpAxis              = &MpAxisBasic_Axis_XM;
	Axis_XM_SMC_PAD.MpAxisParType       = &MpAxis_Axis_XM_ParType;
	Axis_XM_SMC_PAD.MpAxisCyclic        = &MpAxisCyclicSet_Axis_XM;
	Axis_XM_SMC_PAD.MpAxisCyclicParType = &AxisCyclicPar_Axis_XM;
	// Set parameter
	Axis_XM_SMC_PAD.Absolute_Position 				= Axis_XM_HOME_ABSOLUTE_POS;
	Axis_XM_SMC_PAD.Default_parameters.MAX_POSITION = 4000;
	Axis_XM_SMC_PAD.Default_parameters.MIN_POSITION = 0;
	Axis_XM_SMC_PAD.Default_parameters.MAX_VELOCITY = 8000;
	Axis_XM_SMC_PAD.Default_parameters.MIN_VELOCITY = 100;
	// Enable Function block
	Axis_XM_SMC_PAD.Enable = 1;
}

void _CYCLIC ProgramCyclic(void)
{
	switch(dT_Main.xyz_manipulator.X.actual_state){
		case LINP_CTRL_WAIT_STATE:
			{
				if(dT_Main.xyz_manipulator.X.start == 1 && (Axis_XM_SMC_PAD.PowerOn == 1 && Axis_XM_SMC_PAD.IsHomed == 1)){
					dT_Main.xyz_manipulator.X.actual_state = LINP_CTRL_LOAD_PARAM_STATE;
				}
			}
			break;
		case LINP_CTRL_LOAD_PARAM_STATE:
			{
				Axis_XM_SMC_PAD.Set_Parameters.position = Axis_XM_SMC_PAD.Actual_Parameters.position;
				Axis_XM_SMC_PAD.Set_Parameters.velocity = dT_Main.xyz_manipulator.X.parameter.vel;

				Axis_XM_SMC_PAD.Mode.automatic.instruction = INSTR_REAL_TIME;
				Axis_XM_SMC_PAD.Mode.automatic.start = 1;

				dT_Main.xyz_manipulator.X.start = 0;

				if(Axis_XM_SMC_PAD.Internal.State == AUTO_MODE_STATE_RT_1){
					dT_Main.xyz_manipulator.X.actual_state = LINP_CTRL_SET_POSITION_STATE;
				}
			}
			break;
		case LINP_CTRL_SET_POSITION_STATE:
			{
				if(dT_Main.xyz_manipulator.X.stop == 1){
					dT_Main.xyz_manipulator.X.actual_state = LINP_CTRL_STOP_STATE;
				}

				Axis_XM_SMC_PAD.Mode.automatic.start = 0;

				Axis_XM_SMC_PAD.Set_Parameters.velocity = dT_Main.xyz_manipulator.X.parameter.vel;
				Axis_XM_SMC_PAD.Set_Parameters.position = dT_Main.xyz_manipulator.X.parameter.pos;

				dT_Main.xyz_manipulator.X.actual_position = Axis_XM_SMC_PAD.Actual_Parameters.position;
				dT_Main.xyz_manipulator.X.actual_velocity = Axis_XM_SMC_PAD.Actual_Parameters.velocity;
			}
			break;
		case LINP_CTRL_STOP_STATE:
			{
				dT_Main.xyz_manipulator.X.stop = 0;

				Axis_XM_SMC_PAD.Mode.stop = 1;

				if(Axis_XM_SMC_PAD.Internal.State == WAIT_STATE){
					dT_Main.xyz_manipulator.X.actual_state = LINP_CTRL_WAIT_STATE;
				}
			}
			break;
	}

	// Read Data from Main Control Program (Axis inputs)
	Axis_XM_SMC_PAD.Power = dT_Main.service.power;
	Axis_XM_SMC_PAD.Home  = dT_Main.service.home;
	// Write Data to Main Control Program (Information about axis outputs)
	dT_Main.xyz_manipulator.X.active   = Axis_XM_SMC_PAD.Active;
	dT_Main.xyz_manipulator.X.power_on = Axis_XM_SMC_PAD.PowerOn;
	dT_Main.xyz_manipulator.X.is_homed = Axis_XM_SMC_PAD.IsHomed;

	// -------------------- CALL FUNCTION -------------------- //
	// MpAxis - Camera Conveyor AXIS //
	MpAxisBasic(&MpAxisBasic_Axis_XM);
	// MpAxisCyclicSet - Camera Conveyor AXIS //
	MpAxisCyclicSet(&MpAxisCyclicSet_Axis_XM);
	// SMC PAD - Camera Conveyor AXIS //
	SMC_PAD(&Axis_XM_SMC_PAD);
}
```

### Program Logical/XYZ_MANIPULATOR/Y_AXIS_M (ANSIC)

#### Main.c
```c
/**
 * MIT License
 * Copyright(c) 2020 Roman Parak
 * Permission is hereby granted, free of charge, to any person obtaining a copy
 * of this software and associated documentation files (the "Software"), to deal
 * in the Software without restriction, including without limitation the rights
 * to use, copy, modify, merge, publish, distribute, sublicense, and/or sell
 * copies of the Software, and to permit persons to whom the Software is
 * furnished to do so, subject to the following conditions:
 * The above copyright notice and this permission notice shall be included in all
 * copies or substantial portions of the Software.
 * THE SOFTWARE IS PROVIDED "AS IS", WITHOUT WARRANTY OF ANY KIND, EXPRESS OR
 * IMPLIED, INCLUDING BUT NOT LIMITED TO THE WARRANTIES OF MERCHANTABILITY,
 * FITNESS FOR A PARTICULAR PURPOSE AND NONINFRINGEMENT. IN NO EVENT SHALL THE
 * AUTHORS OR COPYRIGHT HOLDERS BE LIABLE FOR ANY CLAIM, DAMAGES OR OTHER
 * LIABILITY, WHETHER IN AN ACTION OF CONTRACT, TORT OR OTHERWISE, ARISING FROM,
 * OUT OF OR IN CONNECTION WITH THE SOFTWARE OR THE USE OR OTHER DEALINGS IN THE
 * SOFTWARE.
 */
/**
 * Author   : Roman Parak
 * Email    : Roman.Parak@outlook.com
 * File Name: Main.c
 */

#include <bur/plc.h>
#include <bur/plctypes.h>
#include "rp_funcx.h"

#ifdef _DEFAULT_INCLUDES
#include <AsDefault.h>
#endif

// {DEFINE - ABSOLUTE POSITION (Camera Conveyor AXIS}
#define Axis_YM_HOME_ABSOLUTE_POS 17700410;
// Camera Conveyor AXIS// MpAxis // STRUCT //
// {Camera Conveyor AXIS}
_LOCAL struct MpAxisBasic MpAxisBasic_Axis_YM;
_LOCAL struct MpAxisBasicParType MpAxis_Axis_YM_ParType;
// {Camera Conveyor AXIS}
_LOCAL struct MpAxisCyclicSet MpAxisCyclicSet_Axis_YM;
_LOCAL struct MpAxisCyclicSetParType AxisCyclicPar_Axis_YM;
// Camera Conveyor AXIS // SMC_PAD // STRUCT //
_LOCAL struct SMC_PAD Axis_YM_SMC_PAD;

void _INIT ProgramInit(void)
{
	// -------------------- INITIALIZATION MAPP AXIS -------------------- //
	// MpAxis SMC PAD //
	MpAxisBasic_Axis_YM.Enable         = 1;
	MpAxisBasic_Axis_YM.Axis           = &gAxis01_Y;
	MpAxisBasic_Axis_YM.MpLink         = &gAxisBasic_Axis_M_Y;
	MpAxisBasic_Axis_YM.Parameters     = &MpAxis_Axis_YM_ParType;
	// Cyclic Parameters {Read}
	MpAxis_Axis_YM_ParType.CyclicRead.MotorTempMode = mpAXIS_READ_CYCLIC;
	MpAxis_Axis_YM_ParType.CyclicRead.LagErrorMode  = mpAXIS_READ_CYCLIC;
	MpAxis_Axis_YM_ParType.CyclicRead.TorqueMode 	= mpAXIS_READ_CYCLIC;
	// MpAxisCyclicSet SMC PAD //
	MpAxisCyclicSet_Axis_YM.Enable 	= 1;
	MpAxisCyclicSet_Axis_YM.MpLink 	= &gAxisBasic_Axis_M_Y;
	MpAxisCyclicSet_Axis_YM.Parameters = &AxisCyclicPar_Axis_YM;
	// MpAxisCyclicSet Parameters (initial) SMC PAD //
	AxisCyclicPar_Axis_YM.Acceleration            = 5000;
	AxisCyclicPar_Axis_YM.Deceleration            = 5000;
	AxisCyclicPar_Axis_YM.PositionModeMaxVelocity = 5000;

	// -------------------- INITIALIZATION SMCTrak -------------------- //
	// Camera Conveyor //
	// MpAxis & MpAxis Cyclic declaration
	Axis_YM_SMC_PAD.MpAxis              = &MpAxisBasic_Axis_YM;
	Axis_YM_SMC_PAD.MpAxisParType       = &MpAxis_Axis_YM_ParType;
	Axis_YM_SMC_PAD.MpAxisCyclic        = &MpAxisCyclicSet_Axis_YM;
	Axis_YM_SMC_PAD.MpAxisCyclicParType = &AxisCyclicPar_Axis_YM;
	// Set parameter
	Axis_YM_SMC_PAD.Absolute_Position 				= Axis_YM_HOME_ABSOLUTE_POS;
	Axis_YM_SMC_PAD.Default_parameters.MAX_POSITION = 5400;
	Axis_YM_SMC_PAD.Default_parameters.MIN_POSITION = 0;
	Axis_YM_SMC_PAD.Default_parameters.MAX_VELOCITY = 8000;
	Axis_YM_SMC_PAD.Default_parameters.MIN_VELOCITY = 100;
	// Enable Function block
	Axis_YM_SMC_PAD.Enable = 1;
}

void _CYCLIC ProgramCyclic(void)
{
	switch(dT_Main.xyz_manipulator.Y.actual_state){
		case LINP_CTRL_WAIT_STATE:
			{
				if(dT_Main.xyz_manipulator.Y.start == 1 && (Axis_YM_SMC_PAD.PowerOn == 1 && Axis_YM_SMC_PAD.IsHomed == 1)){
					dT_Main.xyz_manipulator.Y.actual_state = LINP_CTRL_LOAD_PARAM_STATE;
				}
			}
			break;
		case LINP_CTRL_LOAD_PARAM_STATE:
			{
				Axis_YM_SMC_PAD.Set_Parameters.position = Axis_YM_SMC_PAD.Actual_Parameters.position;
				Axis_YM_SMC_PAD.Set_Parameters.velocity = dT_Main.xyz_manipulator.Y.parameter.vel;

				Axis_YM_SMC_PAD.Mode.automatic.instruction = INSTR_REAL_TIME;
				Axis_YM_SMC_PAD.Mode.automatic.start = 1;

				dT_Main.xyz_manipulator.Y.start = 0;

				if(Axis_YM_SMC_PAD.Internal.State == AUTO_MODE_STATE_RT_1){
					dT_Main.xyz_manipulator.Y.actual_state = LINP_CTRL_SET_POSITION_STATE;
				}
			}
			break;
		case LINP_CTRL_SET_POSITION_STATE:
			{
				if(dT_Main.xyz_manipulator.Y.stop == 1){
					dT_Main.xyz_manipulator.Y.actual_state = LINP_CTRL_STOP_STATE;
				}

				Axis_YM_SMC_PAD.Mode.automatic.start = 0;

				Axis_YM_SMC_PAD.Set_Parameters.velocity = dT_Main.xyz_manipulator.Y.parameter.vel;
				Axis_YM_SMC_PAD.Set_Parameters.position = dT_Main.xyz_manipulator.Y.parameter.pos;

				dT_Main.xyz_manipulator.Y.actual_position = Axis_YM_SMC_PAD.Actual_Parameters.position;
				dT_Main.xyz_manipulator.Y.actual_velocity = Axis_YM_SMC_PAD.Actual_Parameters.velocity;
			}
			break;
		case LINP_CTRL_STOP_STATE:
			{
				dT_Main.xyz_manipulator.Y.stop = 0;

				Axis_YM_SMC_PAD.Mode.stop = 1;

				if(Axis_YM_SMC_PAD.Internal.State == WAIT_STATE){
					dT_Main.xyz_manipulator.Y.actual_state = LINP_CTRL_WAIT_STATE;
				}
			}
			break;
	}

	// Read Data from Main Control Program (Axis inputs)
	Axis_YM_SMC_PAD.Power = dT_Main.service.power;
	Axis_YM_SMC_PAD.Home  = dT_Main.service.home;
	// Write Data to Main Control Program (Information about axis outputs)
	dT_Main.xyz_manipulator.Y.active   = Axis_YM_SMC_PAD.Active;
	dT_Main.xyz_manipulator.Y.power_on = Axis_YM_SMC_PAD.PowerOn;
	dT_Main.xyz_manipulator.Y.is_homed = Axis_YM_SMC_PAD.IsHomed;

	// -------------------- CALL FUNCTION -------------------- //
	// MpAxis - Camera Conveyor AXIS //
	MpAxisBasic(&MpAxisBasic_Axis_YM);
	// MpAxisCyclicSet - Camera Conveyor AXIS //
	MpAxisCyclicSet(&MpAxisCyclicSet_Axis_YM);
	// SMC PAD - Camera Conveyor AXIS //
	SMC_PAD(&Axis_YM_SMC_PAD);
}
```

### Program Logical/XYZ_MANIPULATOR/Z_AXIS_M (ANSIC)
